SYMBOL_TABLE
"SYS_CBitDB"	DB 2	DB 2	// SYS: Changebit interface
"SYS_DirectCtrlDB"	DB 3	DB 3	// GCS7: PC direct control interface default DB
"SYS_HornDB"	DB 4	DB 4	// GCS7: Data Horn Modul
"SYS_LOG_Queue"	DB 5	DB 5	// PC Interface to log
"GCS7_GrCtrlDBTmp"	DB 6	FB 9	// Class date of FB9
"GCS7_RS485CtrlDB"	DB 7	FB 7	// GCS7: Communication controller opto22
"GCS7_ScaleControlDB"	DB 8	DB 8	// GCS7: Scale control buffer
"GCS7_GrCtrlDB"	DB 9	DB 9	// GCS7: Group control buffer
"SYS_DirectCtrlLCDB"	DB 10	DB 10	// GCS7: PC Direct Control Interface Remote Parameter
"TEST_IOSimuliInput"	DB 16	DB 16	// TEST: Only for serial (MPI) simulation
"TEST_IOSimuliOutput"	DB 17	DB 17	// TEST: Only for serial (MPI) simulation
"KebaHT4Data"	DB 20	FB 80	// Data KebaHT4Data
"SYS_PCCDirectCtrlDB"	DB 40	DB 40	// SYS: PC direct control interface PIC / WinCos /MELE
"SYS_PC1DirectCtrlDB"	DB 41	DB 41	// SYS: PC direct control interface pcc 1 (WinCC)
"SYS_PC2DirectCtrlDB"	DB 42	DB 42	// SYS: PC direct control interface pcc 2 (WinCC)
"SYS_PC3DirectCtrlDB"	DB 43	DB 43	// SYS: PC direct control interface pcc 1 (WinCC)
"SYS_PC4DirectCtrlDB"	DB 44	DB 44	// SYS: PC direct control interface pcc 4 (WinCC)
"SYS_PC5DirectCtrlDB"	DB 45	DB 45	// SYS: PC direct control interface pcc 5 (WinCC)
"SYS_PC6DirectCtrlDB"	DB 46	DB 46	// SYS: PC direct control interface pcc 6 (WinCC)
"SYS_PC7DirectCtrlDB"	DB 47	DB 47	// SYS: PC direct control interface pcc 7 (WinCC)
"SYS_ObjViewDirectCtrlDB"	DB 48	DB 48	// SYS: PC direct control interface for ObjView
"SYS_IHTestDirectCtrlDB"	DB 49	DB 49	// SYS: PC direct control interface for inhouse test
"PLC_SystemDB"	DB 50	DB 50	// PLC: System informations
"PLC_DPInfo"	DB 51	DB 51	// Summary Slave errors
"SSA_SYS_ASI_Info"	DB 52	DB 52	// Summary Slave errors
"PC_StorageDB"	DB 53	DB 53	// PC: Storage with free assignment
"ASW_TimerSettings"	DB 56	DB 56	// ASW: Timer settings
"ASW_Counter"	DB 57	DB 57	// ASW: Counter presettings
"SYS_PC1CBitDB"	DB 61	UDT 10020	// SYS: Changebit interface pcc 1 | PIC.LCT | MELE
"SYS_PC2CBitDB"	DB 62	UDT 10020	// SYS: Changebit interface pcc 2 | PIC.LMX
"SYS_PC3CBitDB"	DB 63	UDT 10020	// SYS: Changebit interface pcc 3
"SYS_PC4CBitDB"	DB 64	UDT 10020	// SYS: Changebit interface pcc 4
"GCS7_EREDB"	DB 71	FB 71	// GCS7: ERE
"SYS_DPInfoM1"	DB 75	FB 76	// SYS: PROFIBUS-DP diagnostic master 1
"SYS_DPInfoM2"	DB 76	FB 76	// SYS: PROFIBUS-DP diagnostic master 2
"SYS_DPInfoM3"	DB 77	FB 76	// SYS: PROFIBUS-DP diagnostic master 3
"SYS_DPInfoM4"	DB 78	FB 76	// SYS: PROFIBUS-DP diagnostic master 4
"PLC_BinListDB"	DB 79	FB 79	// Central bin list DB
"ASW_GraphicData"	DB 80	DB 80
"ASW_PlantParData"	DB 81	DB 81	// Plant parameters and data time
"PCC_Data4"	DB 84	DB 84	// WinCC/PIC
"PCC_Data5"	DB 85	DB 85	// WinCC/PIC
"PCC_Data6"	DB 86	DB 86	// WinCC/PIC
"PCC_Data7"	DB 87	DB 87	// WinCC/PIC
"PCC_Data8"	DB 88	DB 88	// WinCC/PIC
"PCC_Data9"	DB 89	DB 89	// WinCC/PIC
"PCC_YieldScaleDB"	DB 90	DB 90	// PCC: Databuffer for PCC yield calculation
"COM_RS485Loop1DB"	DB 91	FB 7	// COM: RS485 loop1 scales and MYEB
"COM_RS485Loop2DB"	DB 92	FB 7	// COM: RS485 loop2 roolers
"COM_RS485Loop3DB"	DB 93	FB 7	// COM: RS485 loop3
"COM_RS485Loop4DB"	DB 94	FB 7	// COM: RS485 loop4
"SYS_SimpleDPInfo4DB"	DB 98	DB 98	// Data DP Diagnose
"SYS_StartWarningDB"	DB 100	FB 100	// SYS:  Startwarning modul
"G001G"	DB 101	FB 101	// Group-DB  Power supply circuit +C11
"G002G"	DB 102	FB 102	// Group-DB  Contactor panel power supply 1
"G003G"	DB 103	FB 103	// Group-DB  PLC monitoring
"G004G"	DB 104	FB 104	// Group-DB  GENERAL ELEMENTS STEEPING
"G005G"	DB 105	FB 105	// Group-DB  GENERAL ELEMENTS GERM 1
"G006G"	DB 106	FB 106	// Group-DB  GENERAL ELEMENTS GERM 2
"G007G"	DB 107	FB 107	// Group-DB  GENERAL ELEMENTS GERM 3
"G008G"	DB 108	FB 108	// Group-DB  GENERAL ELEMENTS GERM 4
"G009G"	DB 109	FB 109	// Group-DB  GENERAL ELEMENTS GERM 5
"G010G"	DB 110	FB 110	// Group-DB  Line messages
"G011G"	DB 111	FB 111	// Group-DB  MELE/WinCoS communication monitoring
"G012G"	DB 112	FB 112	// Group-DB  GENERAL ELEMENTS GERM 6
"G013G"	DB 113	FB 113	// Group-DB  GENERAL ELEMENTS GERM 7
"G014G"	DB 114	FB 114	// Group-DB  GENERAL ELEMENTS GERM 8
"G015G"	DB 115	FB 115	// Group-DB  CCOMPRESSED AIR PRESSURE STEEP 1 - 4
"G016G"	DB 116	FB 116	// Group-DB  CCOMPRESSED AIR PRESSURE STEEP 5 - 8
"G017G"	DB 117	FB 117	// Group-DB  CCOMPRESSED AIR PRESSURE STEEP 9 - 12
"G018G"	DB 118	FB 118	// Group-DB  CCOMPRESSED AIR PRESSURE STEEP 13 - 16
"G019G"	DB 119	FB 119	// Group-DB  CCOMPRESSED AIR PRESSURE STEEP 17 - 20
"G020G"	DB 120	FB 120	// Group-DB  CCOMPRESSED AIR PRESSURE STEEP 21 - 24
"G021G"	DB 121	FB 121	// Group-DB  GENERAL ELEMENTS KILN 1
"G022G"	DB 122	FB 122	// Group-DB  GENERAL ELEMENTS KILN 2
"G023G"	DB 123	FB 123	// Group-DB  GENERAL ELEMENTS KILN MALT TRANSFER
"G026G"	DB 126	FB 126	// Group-DB  Alarm horns
"G029G"	DB 129	FB 129	// Group-DB  Bin low levels
"G030G"	DB 130	FB 130	// Group-DB  Bin high levels
"G031G"	DB 131	FB 131	// Group-DB  GENERAL ELEMENTS STEEPING
"G032M"	DB 132	FB 132	// Group-DB  CO2 FAN AND FESH AIR FLAP STEEPING 1
"G033M"	DB 133	FB 133	// Group-DB  AERATION AIR STEEPING 1
"G034M"	DB 134	FB 134	// Group-DB  CO2 FAN AND FESH AIR FLAP STEEPING 2
"G035M"	DB 135	FB 135	// Group-DB  AERATION AIR STEEPING 2
"G036M"	DB 136	FB 136	// Group-DB  CO2 FAN AND FESH AIR FLAP STEEPING 3
"G037M"	DB 137	FB 137	// Group-DB  AERATION AIR STEEPING 3
"G038M"	DB 138	FB 138	// Group-DB  CO2 FAN AND FESH AIR FLAP STEEPING 4
"G039M"	DB 139	FB 139	// Group-DB  AERATION AIR STEEPING 4
"G040M"	DB 140	FB 140	// Group-DB  CO2 FAN AND FESH AIR FLAP STEEPING 5
"G041M"	DB 141	FB 141	// Group-DB  AERATION AIR STEEPING 5
"G042M"	DB 142	FB 142	// Group-DB  CO2 FAN AND FESH AIR FLAP STEEPING 6
"G043M"	DB 143	FB 143	// Group-DB  AERATION AIR STEEPING 6
"G044M"	DB 144	FB 144	// Group-DB  CO2 FAN AND FESH AIR FLAP STEEPING 7
"G045M"	DB 145	FB 145	// Group-DB  AERATION AIR STEEPING 7
"G046M"	DB 146	FB 146	// Group-DB  CO2 FAN AND FESH AIR FLAP STEEPING 8
"G047M"	DB 147	FB 147	// Group-DB  AERATION AIR STEEPING 8
"G048M"	DB 148	FB 148	// Group-DB  CO2 FAN AND FESH AIR FLAP STEEPING 9
"G049M"	DB 149	FB 149	// Group-DB  AERATION AIR STEEPING 9
"G050M"	DB 150	FB 150	// Group-DB  CO2 FAN AND FESH AIR FLAP STEEPING 10
"G051M"	DB 151	FB 151	// Group-DB  AERATION AIR STEEPING 10
"G052M"	DB 152	FB 152	// Group-DB  CO2 FAN AND FESH AIR FLAP STEEPING 11
"G053M"	DB 153	FB 153	// Group-DB  AERATION AIR STEEPING 11
"G054M"	DB 154	FB 154	// Group-DB  CO2 FAN AND FESH AIR FLAP STEEPING 12
"G055M"	DB 155	FB 155	// Group-DB  AERATION AIR STEEPING 12
"G056M"	DB 156	FB 156	// Group-DB  CO2 FAN AND FESH AIR FLAP STEEPING 13
"G057M"	DB 157	FB 157	// Group-DB  AERATION AIR STEEPING 13
"G058M"	DB 158	FB 158	// Group-DB  CO2 FAN AND FESH AIR FLAP STEEPING 14
"G059M"	DB 159	FB 159	// Group-DB  AERATION AIR STEEPING 14
"G060M"	DB 160	FB 160	// Group-DB  CO2 FAN AND FESH AIR FLAP STEEPING 15
"G061M"	DB 161	FB 161	// Group-DB  AERATION AIR STEEPING 15
"G062M"	DB 162	FB 162	// Group-DB  CO2 FAN AND FESH AIR FLAP STEEPING 16
"G063M"	DB 163	FB 163	// Group-DB  AERATION AIR STEEPING 16
"G064M"	DB 164	FB 164	// Group-DB  CO2 FAN AND FESH AIR FLAP STEEPING 17
"G065M"	DB 165	FB 165	// Group-DB  AERATION AIR STEEPING 17
"G066M"	DB 166	FB 166	// Group-DB  PRODUCT SLIDER STEEPING 17
"G067M"	DB 167	FB 167	// Group-DB  CO2 FAN AND FESH AIR FLAP STEEPING 18
"G068M"	DB 168	FB 168	// Group-DB  AERATION AIR STEEPING 18
"G069M"	DB 169	FB 169	// Group-DB  PRODUCT SLIDER STEEPING 18
"G070M"	DB 170	FB 170	// Group-DB  CO2 FAN AND FESH AIR FLAP STEEPING 19
"G071M"	DB 171	FB 171	// Group-DB  AERATION AIR STEEPING 19
"G072M"	DB 172	FB 172	// Group-DB  PRODUCT SLIDER STEEPING 19
"G073M"	DB 173	FB 173	// Group-DB  CO2 FAN AND FESH AIR FLAP STEEPING 20
"G074M"	DB 174	FB 174	// Group-DB  AERATION AIR STEEPING 20
"G075M"	DB 175	FB 175	// Group-DB  PRODUCT SLIDER STEEPING 20
"G076M"	DB 176	FB 176	// Group-DB  CO2 FAN AND FESH AIR FLAP STEEPING 21
"G077M"	DB 177	FB 177	// Group-DB  AERATION AIR STEEPING 21
"G078M"	DB 178	FB 178	// Group-DB  PRODUCT SLIDER STEEPING 21
"G079M"	DB 179	FB 179	// Group-DB  CO2 FAN AND FESH AIR FLAP STEEPING 22
"G080M"	DB 180	FB 180	// Group-DB  AERATION AIR STEEPING 22
"G081M"	DB 181	FB 181	// Group-DB  PRODUCT SLIDER STEEPING 22
"G082M"	DB 182	FB 182	// Group-DB  CO2 FAN AND FESH AIR FLAP STEEPING 23
"G083M"	DB 183	FB 183	// Group-DB  AERATION AIR STEEPING 23
"G084M"	DB 184	FB 184	// Group-DB  PRODUCT SLIDER STEEPING 23
"G085M"	DB 185	FB 185	// Group-DB  CO2 FAN AND FESH AIR FLAP STEEPING 24
"G086M"	DB 186	FB 186	// Group-DB  AERATION AIR STEEPING 24
"G087M"	DB 187	FB 187	// Group-DB  PRODUCT SLIDER STEEPING 24
"G090G"	DB 190	FB 190	// Group-DB  GENERAL ELEMENTS GERM 1
"G091M"	DB 191	FB 191	// Group-DB  BELT CONVEYOR 4100 GERM 1-4
"G092M"	DB 192	FB 192	// Group-DB  BELT CONVEYOR 4200 GERM 5-8
"G093M"	DB 193	FB 193	// Group-DB  BELT CONVEYOR 4300 GERM
"G094M"	DB 194	FB 194	// Group-DB  BELT CONVEYOR 4400 GERM
"G095M"	DB 195	FB 195	// Group-DB  BELT CONVEYOR 4500 GERM
"G097M"	DB 197	FB 197	// Group-DB  LIFTING DEVICE GERM 1
"G098M"	DB 198	FB 198	// Group-DB  COUPLING DEVICE TURNER GERM 1
"G099M"	DB 199	FB 199	// Group-DB  COUPLING DEVICE WALL GERM 1
"G100M"	DB 200	FB 200	// Group-DB  TRAVELLING DRIVE GERM 1
"G101M"	DB 201	FB 201	// Group-DB  HORIZONTAL AND LIFTING SCREW GERM 1
"G102M"	DB 202	FB 202	// Group-DB  LOCAL COMMAND BUTTON / LAMPS GERM 1
"G103M"	DB 203	FB 203	// Group-DB  TEMPERATURE MES. GERM 1
"G104M"	DB 204	FB 204	// Group-DB  TURNING SCREWS GERM 1
"G105M"	DB 205	FB 205	// Group-DB  FAN AND VALVE SRAY AIR GERM 1
"G106M"	DB 206	FB 206	// Group-DB  FRESH AIR LOUVER GERM 1
"G107M"	DB 207	FB 207	// Group-DB  EXHAUST AIR LOUVER GERM 1
"G108M"	DB 208	FB 208	// Group-DB  PRODUCT MOISTERING  GERM 1
"G109M"	DB 209	FB 209	// Group-DB  HP CLEANING GERM 1
"G110M"	DB 210	FB 210	// Group-DB  INLET SLIDE GERM 1
"G111M"	DB 211	FB 211	// Group-DB  LOADING CONVEYOR 4600 GERM 1
"G112M"	DB 212	FB 212	// Group-DB  COOLING / HEATING GERM 1
"G113M"	DB 213	FB 213	// Group-DB  BELT CONVEYOR 7050 GERM 1 / 2
"G114M"	DB 214	FB 214	// Group-DB  CHAIN CONVEYOR 7100 GERM
"G120G"	DB 220	FB 220	// Group-DB  GENERAL ELEMENTS GERM 2
"G121M"	DB 221	FB 221	// Group-DB  CHAIN CONVEYOR 4600 GERM 2
"G122M"	DB 222	FB 222	// Group-DB  LIFTING DEVICE GERM 2
"G123M"	DB 223	FB 223	// Group-DB  COUPLING DEVICE TURNER GERM 2
"G124M"	DB 224	FB 224	// Group-DB  COUPLING DEVICE WALL GERM 2
"G125M"	DB 225	FB 225	// Group-DB  TRAVELLING DRIVE GERM 2
"G126M"	DB 226	FB 226	// Group-DB  HORIZONTAL AND LIFTING SCREW GERM 2
"G127M"	DB 227	FB 227	// Group-DB  LOCAL COMMAND BUTTON / LAMPS GERM 2
"G128M"	DB 228	FB 228	// Group-DB  TEMPERATURE MES. GERM 2
"G129M"	DB 229	FB 229	// Group-DB  TURNING SCREWS GERM 2
"G130M"	DB 230	FB 230	// Group-DB  FAN AND VALVE SRAY AIR GERM 2
"G131M"	DB 231	FB 231	// Group-DB  FRESH AIR LOUVER GERM 2
"G132M"	DB 232	FB 232	// Group-DB  EXHAUST AIR  LOUVER GERM 2
"G133M"	DB 233	FB 233	// Group-DB  PRODUCT MOISTERING  GERM 2
"G134M"	DB 234	FB 234	// Group-DB  HP CLEANING GERM 2
"G135M"	DB 235	FB 235	// Group-DB  INLET SLIDE GERM 2
"G136M"	DB 236	FB 236	// Group-DB  LOAD / UNLOAD CONVEYOR GERM 2
"G137M"	DB 237	FB 237	// Group-DB  COOLING / HEATING GERM 2
"G140G"	DB 240	FB 240	// Group-DB  GENERAL ELEMENTS GERM 3
"G141M"	DB 241	FB 241	// Group-DB  CHAIN CONVEYOR 4600 GERM 3
"G142M"	DB 242	FB 242	// Group-DB  LIFTING DEVICE GERM 3
"G143M"	DB 243	FB 243	// Group-DB  COUPLING DEVICE TURNER GERM 3
"G144M"	DB 244	FB 244	// Group-DB  COUPLING DEVICE WALL GERM 3
"G145M"	DB 245	FB 245	// Group-DB  TRAVELLING DRIVE GERM 3
"G146M"	DB 246	FB 246	// Group-DB  HORIZONTAL AND LIFTING SCREW GERM 3
"G147M"	DB 247	FB 247	// Group-DB  LOCAL COMMAND BUTTON / LAMPS GERM 3
"G148M"	DB 248	FB 248	// Group-DB  TEMPERATURE MES. GERM 3
"G149M"	DB 249	FB 249	// Group-DB  TURNING SCREWS GERM 3
"G150M"	DB 250	FB 250	// Group-DB  FAN AND VALVE SRAY AIR GERM 3
"G151M"	DB 251	FB 251	// Group-DB  FRESH AIR LOUVER GERM 3
"G152M"	DB 252	FB 252	// Group-DB  EXHAUST AIR LOUVER GERM 3
"G153M"	DB 253	FB 253	// Group-DB  PRODUCT MOISTERING  GERM 3
"G154M"	DB 254	FB 254	// Group-DB  HP CLEANING GERM 3
"G155M"	DB 255	FB 255	// Group-DB  INLET SLIDE GERM 3
"G156M"	DB 256	FB 256	// Group-DB  LOAD / UNLOAD CONVEYOR GERM 3
"G157M"	DB 257	FB 257	// Group-DB  COOLING / HEATING GERM 3
"G158M"	DB 258	FB 258	// Group-DB  CHAIN CONVEYOR 7050 GERM 3 / 4
"G160G"	DB 260	FB 260	// Group-DB  GENERAL ELEMENTS GERM 4
"G161M"	DB 261	FB 261	// Group-DB  CHAIN CONVEYOR 4600 GERM 4
"G162M"	DB 262	FB 262	// Group-DB  LIFTING DEVICE GERM 4
"G163M"	DB 263	FB 263	// Group-DB  COUPLING DEVICE TURNER GERM 4
"G164M"	DB 264	FB 264	// Group-DB  COUPLING DEVICE WALL GERM 4
"G165M"	DB 265	FB 265	// Group-DB  TRAVELLING DRIVE GERM 4
"G166M"	DB 266	FB 266	// Group-DB  HORIZONTAL AND LIFTING SCREW GERM 4
"G167M"	DB 267	FB 267	// Group-DB  LOCAL COMMAND BUTTON / LAMPS GERM 4
"G168M"	DB 268	FB 268	// Group-DB  TEMPERATURE MES. GERM 4
"G169M"	DB 269	FB 269	// Group-DB  TURNING SCREWS GERM 4
"G170M"	DB 270	FB 270	// Group-DB  FAN AND VALVE SRAY AIR GERM 4
"G171M"	DB 271	FB 271	// Group-DB  FRESH AIR LOUVER GERM 4
"G172M"	DB 272	FB 272	// Group-DB  EXHAUST AIR LOUVER GERM 4
"G173M"	DB 273	FB 273	// Group-DB  PRODUCT MOISTERING  GERM 4
"G174M"	DB 274	FB 274	// Group-DB  HP CLEANING GERM 4
"G175M"	DB 275	FB 275	// Group-DB  INLET SLIDE GERM 4
"G176M"	DB 276	FB 276	// Group-DB  LOAD / UNLOAD CONVEYOR GERM 4
"G177M"	DB 277	FB 277	// Group-DB  COOLING / HEATING GERM 4
"G180G"	DB 280	FB 280	// Group-DB  GENERAL ELEMENTS GERM 5
"G181M"	DB 281	FB 281	// Group-DB  CHAIN CONVEYOR 4600 GERM 5
"G182M"	DB 282	FB 282	// Group-DB  LIFTING DEVICE GERM 5
"G183M"	DB 283	FB 283	// Group-DB  COUPLING DEVICE TURNER GERM 5
"G184M"	DB 284	FB 284	// Group-DB  COUPLING DEVICE WALL GERM 5
"G185M"	DB 285	FB 285	// Group-DB  TRAVELLING DRIVE GERM 5
"G186M"	DB 286	FB 286	// Group-DB  HORIZONTAL AND LIFTING SCREW GERM 5
"G187M"	DB 287	FB 287	// Group-DB  LOCAL COMMAND BUTTON / LAMPS GERM 5
"G188M"	DB 288	FB 288	// Group-DB  TEMPERATURE MES. GERM 5
"G189M"	DB 289	FB 289	// Group-DB  TURNING SCREWS GERM 5
"G190M"	DB 290	FB 290	// Group-DB  FAN AND VALVE SRAY AIR GERM 5
"G191M"	DB 291	FB 291	// Group-DB  FRESH AIR LOUVER GERM 5
"G192M"	DB 292	FB 292	// Group-DB  EXHAUST AIR LOUVER GERM 5
"G193M"	DB 293	FB 293	// Group-DB  PRODUCT MOISTERING  GERM 5
"G194M"	DB 294	FB 294	// Group-DB  HP CLEANING GERM 5
"G195M"	DB 295	FB 295	// Group-DB  INLET SLIDE GERM 5
"G196M"	DB 296	FB 296	// Group-DB  LOAD / UNLOAD CONVEYOR GERM 5
"G197M"	DB 297	FB 297	// Group-DB  COOLING / HEATING GERM 5
"G198M"	DB 298	FB 298	// Group-DB  CHAIN CONVEYOR 7050 GERM 5 / 6
"G200G"	DB 300	FB 300	// Group-DB  GENERAL ELEMENTS GERM 6
"G201M"	DB 301	FB 301	// Group-DB  CHAIN CONVEYOR 4600 GERM 6
"G202M"	DB 302	FB 302	// Group-DB  LIFTING DEVICE GERM 6
"G203M"	DB 303	FB 303	// Group-DB  COUPLING DEVICE TURNER GERM 6
"G204M"	DB 304	FB 304	// Group-DB  COUPLING DEVICE WALL GERM 6
"G205M"	DB 305	FB 305	// Group-DB  TRAVELLING DRIVE GERM 6
"G206M"	DB 306	FB 306	// Group-DB  HORIZONTAL AND LIFTING SCREW GERM 6
"G207M"	DB 307	FB 307	// Group-DB  LOCAL COMMAND BUTTON / LAMPS GERM 6
"G208M"	DB 308	FB 308	// Group-DB  TEMPERATURE MES. GERM 6
"G209M"	DB 309	FB 309	// Group-DB  TURNING SCREWS GERM 6
"G210M"	DB 310	FB 310	// Group-DB  FAN AND VALVE SRAY AIR GERM 6
"G211M"	DB 311	FB 311	// Group-DB  FRESH AIR LOUVER GERM 6
"G212M"	DB 312	FB 312	// Group-DB  EXHAUST AIR LOUVER GERM 6
"G213M"	DB 313	FB 313	// Group-DB  PRODUCT MOISTERING  GERM 6
"G214M"	DB 314	FB 314	// Group-DB  HP CLEANING GERM 6
"G215M"	DB 315	FB 315	// Group-DB  INLET SLIDE GERM 6
"G216M"	DB 316	FB 316	// Group-DB  LOAD / UNLOAD CONVEYOR GERM 6
"G217M"	DB 317	FB 317	// Group-DB  COOLING / HEATING GERM 6
"G220G"	DB 320	FB 320	// Group-DB  GENERAL ELEMENTS GERM 7
"G221M"	DB 321	FB 321	// Group-DB  CHAIN CONVEYOR 4600 GERM 7
"G222M"	DB 322	FB 322	// Group-DB  LIFTING DEVICE GERM 7
"G223M"	DB 323	FB 323	// Group-DB  COUPLING DEVICE TURNER GERM 7
"G224M"	DB 324	FB 324	// Group-DB  COUPLING DEVICE WALL GERM 7
"G225M"	DB 325	FB 325	// Group-DB  TRAVELLING DRIVE GERM 7
"G226M"	DB 326	FB 326	// Group-DB  HORIZONTAL AND LIFTING SCREW GERM 7
"G227M"	DB 327	FB 327	// Group-DB  LOCAL COMMAND BUTTON / LAMPS GERM 7
"G228M"	DB 328	FB 328	// Group-DB  TEMPERATURE MES. GERM 7
"G229M"	DB 329	FB 329	// Group-DB  TURNING SCREWS GERM 7
"G230M"	DB 330	FB 330	// Group-DB  FAN AND VALVE SRAY AIR GERM 7
"G231M"	DB 331	FB 331	// Group-DB  FRESH AIR LOUVER GERM 7
"G232M"	DB 332	FB 332	// Group-DB  EXHAUST AIR LOUVER GERM 7
"G233M"	DB 333	FB 333	// Group-DB  PRODUCT MOISTERING  GERM 7
"G234M"	DB 334	FB 334	// Group-DB  HP CLEANING GERM 7
"G235M"	DB 335	FB 335	// Group-DB  INLET SLIDE GERM 7
"G236M"	DB 336	FB 336	// Group-DB  LOAD / UNLOAD CONVEYOR GERM 7
"G237M"	DB 337	FB 337	// Group-DB  COOLING / HEATING GERM 7
"G238M"	DB 338	FB 338	// Group-DB  CHAIN CONVEYOR 7050 GERM 7 / 8
"G240G"	DB 340	FB 340	// Group-DB  GENERAL ELEMENTS GERM 8
"G241M"	DB 341	FB 341	// Group-DB  CHAIN CONVEYOR 4600 GERM 8
"G242M"	DB 342	FB 342	// Group-DB  LIFTING DEVICE GERM 8
"G243M"	DB 343	FB 343	// Group-DB  COUPLING DEVICE TURNER GERM 8
"G244M"	DB 344	FB 344	// Group-DB  COUPLING DEVICE WALL GERM 8
"G245M"	DB 345	FB 345	// Group-DB  TRAVELLING DRIVE GERM 8
"G246M"	DB 346	FB 346	// Group-DB  HORIZONTAL AND LIFTING SCREW GERM 8
"G247M"	DB 347	FB 347	// Group-DB  LOCAL COMMAND BUTTON / LAMPS GERM 8
"G248M"	DB 348	FB 348	// Group-DB  TEMPERATURE MES. GERM 8
"G249M"	DB 349	FB 349	// Group-DB  TURNING SCREWS GERM 8
"G250M"	DB 350	FB 350	// Group-DB  FAN AND VALVE SRAY AIR GERM 8
"G251M"	DB 351	FB 351	// Group-DB  FRESH AIR LOUVER GERM 8
"G252M"	DB 352	FB 352	// Group-DB  EXHAUST AIR LOUVER GERM 8
"G253M"	DB 353	FB 353	// Group-DB  PRODUCT MOISTERING  GERM 8
"G254M"	DB 354	FB 354	// Group-DB  HP CLEANING GERM 8
"G255M"	DB 355	FB 355	// Group-DB  INLET SLIDE GERM 8
"G256M"	DB 356	FB 356	// Group-DB  LOAD / UNLOAD CONVEYOR GERM 8
"G257M"	DB 357	FB 357	// Group-DB  COOLING / HEATING GERM 8
"G260G"	DB 360	FB 360	// Group-DB  GENERAL ELEMENTS KILN 1
"G261M"	DB 361	FB 361	// Group-DB  BELT CONVEYOR 7200 KILN
"G262M"	DB 362	FB 362	// Group-DB  BELT CONVEYOR 7300 KILN
"G263M"	DB 363	FB 363	// Group-DB  BELT CONVEYOR 7301 KILN
"G264M"	DB 364	FB 364	// Group-DB  BELT CONVEYOR 7400 KILN
"G265M"	DB 365	FB 365	// Group-DB  LIFTING DEVICE KILN 1
"G266M"	DB 366	FB 366	// Group-DB  TRAVELLING DRIVE KILN 1
"G267M"	DB 367	FB 367	// Group-DB  UNLOADING / LOADING SCREW KILN 1
"G268M"	DB 368	FB 368	// Group-DB  DISCHARGE DOOR KILN 1
"G269M"	DB 369	FB 369	// Group-DB  TEMPERATURE MES. KILN 1
"G270M"	DB 370	FB 370	// Group-DB  AIR SHUT SLIDE KILN 1
"G271M"	DB 371	FB 371	// Group-DB  FAN KILN 1
"G272M"	DB 372	FB 372	// Group-DB  FRESH AIR RECYCLING KILN 1
"G273M"	DB 373	FB 373	// Group-DB  RECYCLING AIR LOUVER KILN 1
"G274M"	DB 374	FB 374	// Group-DB  EXHAUST AIR LOUVER KILN 1
"G275M"	DB 375	FB 375	// Group-DB  BYPASS FLAP KILN 1
"G276M"	DB 376	FB 376	// Group-DB  HEATING KILN 1
"G277M"	DB 377	FB 377	// Group-DB  LOUVER AIR HEATER KILN 1
"G278M"	DB 378	FB 378	// Group-DB  WITHERING AIR KILN 1
"G279M"	DB 379	FB 379	// Group-DB  HEATING KILN 1 + 2
"G280M"	DB 380	FB 380	// Group-DB  CHAIN CONVEYOR 9001 KILN 1
"G281M"	DB 381	FB 381	// Group-DB  ELEVATOR 9002 AFTER KILN
"G282M"	DB 382	FB 382	// Group-DB  FLAP BOX 9008
"G283M"	DB 383	FB 383	// Group-DB  CULM BATCH BIN 9005
"G284M"	DB 384	FB 384	// Group-DB  BELT CONVEYOR 7100 KILN
"G290G"	DB 390	FB 390	// Group-DB  GENERAL ELEMENTS KILN 2
"G291M"	DB 391	FB 391	// Group-DB  LIFTING DEVICE KILN 2
"G292M"	DB 392	FB 392	// Group-DB  TRAVELLING DRIVE KILN 2
"G293M"	DB 393	FB 393	// Group-DB  UNLOADING / LOADING SCREW KILN 2
"G294M"	DB 394	FB 394	// Group-DB  DISCHARGE DOOR KILN 2
"G295M"	DB 395	FB 395	// Group-DB  TEMPERATURE MES. KILN 2
"G296M"	DB 396	FB 396	// Group-DB  AIR SHUT SLIDE KILN 2
"G297M"	DB 397	FB 397	// Group-DB  FAN KILN 2
"G298M"	DB 398	FB 398	// Group-DB  FRESH AIR FLAP KILN 2
"G299M"	DB 399	FB 399	// Group-DB  RECYCLING AIR FLAP KILN 2
"G300M"	DB 400	FB 400	// Group-DB  EXHAUST AIR FLAP KILN 2
"G301M"	DB 401	FB 401	// Group-DB  BYPASS FLAP KILN 2
"G302M"	DB 402	FB 402	// Group-DB  HEATING KILN 2
"G303M"	DB 403	FB 403	// Group-DB  LOUVER AIR HEATER KILN 2
"G304M"	DB 404	FB 404	// Group-DB  WITHERING AIR KILN 2
"G305M"	DB 405	FB 405	// Group-DB  CHAIN CONVEYOR 9002 KILN 2
"G306M"	DB 406	FB 406	// Group-DB  DMBG DISCHARGER KILN MALT TRANSFER
"G307M"	DB 407	FB 407	// Group-DB  SCREW CONVEYOR 9007 KILN MALT TRANSFER
"G308M"	DB 408	FB 408	// Group-DB  BELT CONVEYOR 9009 KILN MALT TRANSFER
"G309M"	DB 409	FB 409	// Group-DB  ELEVATOR EXCISTING
"G310M"	DB 410	FB 410	// Group-DB  PLC1 TO EXCISTING DEGERMINATION SYSTEM
"G311M"	DB 411	FB 411	// Group-DB  CENTRAL ASPIRATION UNLOAD KILN
"G320M"	DB 420	FB 420	// Group-DB  PCC GRAPHIC SUPPORT
"EventsToPIC_DB"	DB 470	FB 470
"ASW_DFCATargData"	DB 480	DB 480	// ASW_DFCATargData
"INT1S001SND33"	DB 515	DB 515	// Bin DB  Wheat intake sender
"INT1S001RCV34"	DB 516	DB 516	// Bin DB  Wheat intake receiver
"FCL1S001SND33"	DB 535	DB 535	// Bin DB  1st cleaning sender
"FCL1S001RCV34"	DB 536	DB 536	// Bin DB  1st cleaning receiver
"SDP1S001SND33"	DB 545	DB 545	// Bin DB  2nd dampening sender
"SDP1S001RCV34"	DB 546	DB 546	// Bin DB  2nd dampening receiver
"SCL1S001SND33"	DB 555	DB 555	// Bin DB  2nd cleaning sender
"SCL1S001RCV34"	DB 556	DB 556	// Bin DB  2nd cleaning receiver
"FTR1S001SND33"	DB 575	DB 575	// Bin DB  Flour transfer sender
"FTR1S001RCV34"	DB 576	DB 576	// Bin DB  Flour transfer receiver
"OTL1S001SND33"	DB 585	DB 585	// Bin DB  Flour bulk outload sender
"OTL1S001RCV34"	DB 586	DB 586	// Bin DB  Flour bulk outload receiver
"SCG1S001SND33"	DB 595	DB 595	// Bin DB  Screenings grinding sender
"SCG1S001RCV34"	DB 596	DB 596	// Bin DB  Screenings grinding receiver
"BTR1S001SND33"	DB 605	DB 605	// Bin DB  Bran turnover sender
"BTR1S001RCV34"	DB 606	DB 606	// Bin DB  Bran turnover receiver
"MAL1Par"	DB 799	DB 799	// Line parameter data block
"MAL1"	DB 800	DB 800	// Line data block  MALTING LINE
"MAL1S001"	DB 801	DB 801	// Section data block  LINE 1 SEC 1 SECTIONDATA
"MAL1S005"	DB 805	DB 805	// Section data block  STEEPING ROW 1 (ST1-8)
"MAL1S006"	DB 806	DB 806	// Section data block  STEEPING ROW 2 (ST9-16)
"MAL1S007"	DB 807	DB 807	// Section data block  STEEPING ROW 3 (ST17-24)
"MAL1S017"	DB 817	DB 817	// Section data block  LINE 1 SEC 17 GERM 1
"MAL1S018"	DB 818	DB 818	// Section data block  LINE 1 SEC 18 GERM 2
"MAL1S019"	DB 819	DB 819	// Section data block  LINE 1 SEC 19 GERM 3
"MAL1S020"	DB 820	DB 820	// Section data block  LINE 1 SEC 20 GERM 4
"MAL1S021"	DB 821	DB 821	// Section data block  LINE 1 SEC 21 GERM 5
"MAL1S022"	DB 822	DB 822	// Section data block  LINE 1 SEC 22 GERM 6
"MAL1S023"	DB 823	DB 823	// Section data block  LINE 1 SEC 23 GERM 7
"MAL1S024"	DB 824	DB 824	// Section data block  LINE 1 SEC 24 GERM 8
"MAL1S032"	DB 832	DB 832	// Section data block  LINE 1 SEC 32 KILN 1
"MAL1S033"	DB 833	DB 833	// Section data block  LINE 1 SEC 33 KILN 2
"MAL1S034"	DB 834	DB 834	// Section data block  LINE 1 SEC 34 UNLOAD KILN
"MAL1S001SND33"	DB 843	DB 843	// Bin DB  Dummy sender
"MAL1S001RCV34"	DB 844	DB 844	// Bin DB  Dummy receiver
"MAl1S034SND35"	DB 845	DB 845	// Bin DB  KILNED MALT BINS
"MAl1S034RCV36"	DB 846	DB 846	// Bin DB  KILNED MALT BINS
"MAL1S005Par"	DB 895	DB 895	// Parameter data block  STEEPING ROW 1 (ST1-8)
"MAL1S006Par"	DB 896	DB 896	// Parameter data block  STEEPING ROW 2 (ST9-16)
"MAL1S007Par"	DB 897	DB 897	// Parameter data block  STEEPING ROW 3 (ST17-24)
"MAL1S005_ST1Par"	DB 900	DB 900	// Parameter data block  STEEPING ROW 1 (ST1-8)
"MAL1S017Par"	DB 907	DB 907	// Parameter data block  LINE 1 SEC 17 GERM 1
"MAL1S018Par"	DB 908	DB 908	// Parameter data block  LINE 1 SEC 18 GERM 2
"MAL1S019Par"	DB 909	DB 909	// Parameter data block  LINE 1 SEC 19 GERM 3
"MAL1S020Par"	DB 910	DB 910	// Parameter data block  LINE 1 SEC 20 GERM 4
"MAL1S021Par"	DB 911	DB 911	// Parameter data block  LINE 1 SEC 21 GERM 5
"MAL1S022Par"	DB 912	DB 912	// Parameter data block  LINE 1 SEC 22 GERM 6
"MAL1S023Par"	DB 913	DB 913	// Parameter data block  LINE 1 SEC 23 GERM 7
"MAL1S024Par"	DB 914	DB 914	// Parameter data block  LINE 1 SEC 24 GERM 8
"MAL1S032Par"	DB 922	DB 922	// Parameter data block  LINE 1 SEC 32 KILN 1
"MAL1S033Par"	DB 923	DB 923	// Parameter data block  LINE 1 SEC 33 KILN 2
"SSA_LOG_Value_Queue"	DB 1005	DB 1005	// PC Interface to log
"MAL1ProcessTime"	DB 1013	DB 1013	// ProcessTime  MALTING LINE
"PLC1Snd"	DB 1711	DB 1711	// COM: Send data to PLC 1
"PLC2Snd"	DB 1712	DB 1712	// COM: Send data to PLC 2
"PLC3Snd"	DB 1713	DB 1713	// COM: Send data to PLC 3
"PLC4Snd"	DB 1714	DB 1714	// COM: Send data to PLC 4
"PLC5Snd"	DB 1715	DB 1715	// COM: Send data to PLC 5
"PLC6Snd"	DB 1716	DB 1716	// COM: Send data to PLC 6
"PLC7Snd"	DB 1717	DB 1717	// COM: Send data to PLC 7
"PLC8Snd"	DB 1718	DB 1718	// COM: Send data to PLC 8
"PLC9Snd"	DB 1719	DB 1719	// COM: Send data to PLC 9
"PLC1Rcv"	DB 1721	DB 1721	// COM: Receive data from PLC 1
"PLC2Rcv"	DB 1722	DB 1722	// COM: Receive data from PLC 2
"PLC3Rcv"	DB 1723	DB 1723	// COM: Receive data from PLC 3
"PLC4Rcv"	DB 1724	DB 1724	// COM: Receive data from PLC 4
"PLC5Rcv"	DB 1725	DB 1725	// COM: Receive data from PLC 5
"PLC6Rcv"	DB 1726	DB 1726	// COM: Receive data from PLC 6
"PLC7Rcv"	DB 1727	DB 1727	// COM: Receive data from PLC 7
"PLC8Rcv"	DB 1728	DB 1728	// COM: Receive data from PLC 8
"PLC9Rcv"	DB 1729	DB 1729	// COM: Receive data from PLC 9
"PLC10Snd"	DB 1730	DB 1730	// COM: Send data to PLC 10
"PLC11Snd"	DB 1731	DB 1731	// COM: Send data to PLC 11
"PLC12Snd"	DB 1732	DB 1732	// COM: Send data to PLC 12
"PLC13Snd"	DB 1733	DB 1733	// COM: Send data to PLC 13
"PLC14Snd"	DB 1734	DB 1734	// COM: Send data to PLC 14
"PLC15Snd"	DB 1735	DB 1735	// COM: Send data to PLC 15
"PLC16Snd"	DB 1736	DB 1736	// COM: Send data to PLC 16
"PLC10Rcv"	DB 1740	DB 1740	// COM: Receive data from PLC 10
"PLC11Rcv"	DB 1741	DB 1741	// COM: Receive data from PLC 11
"PLC12Rcv"	DB 1742	DB 1742	// COM: Receive data from PLC 12
"PLC13Rcv"	DB 1743	DB 1743	// COM: Receive data from PLC 13
"PLC14Rcv"	DB 1744	DB 1744	// COM: Receive data from PLC 14
"PLC15Rcv"	DB 1745	DB 1745	// COM: Receive data from PLC 15
"PLC16Rcv"	DB 1746	DB 1746	// COM: Receive data from PLC 16
"ComPLC1Snd"	DB 1761	FB 1701	// COM: Send buffer PLC 1
"ComPLC2Snd"	DB 1762	FB 1701	// COM: Send buffer PLC 2
"ComPLC3Snd"	DB 1763	FB 1701	// COM: Send buffer PLC 3
"ComPLC4Snd"	DB 1764	FB 1701	// COM: Send buffer PLC 4
"ComPLC5Snd"	DB 1765	FB 1701	// COM: Send buffer PLC 5
"ComPLC6Snd"	DB 1766	FB 1701	// COM: Send buffer PLC 6
"ComPLC7Snd"	DB 1767	FB 1701	// COM: Send buffer PLC 7
"ComPLC8Snd"	DB 1768	FB 1701	// COM: Send buffer PLC 8
"ComPLC9Snd"	DB 1769	FB 1701	// COM: Send buffer PLC 9
"ComPLC1Rcv"	DB 1771	FB 1702	// COM: Receive buffer PLC 1
"ComPLC2Rcv"	DB 1772	FB 1702	// COM: Receive buffer PLC 2
"ComPLC3Rcv"	DB 1773	FB 1702	// COM: Receive buffer PLC 3
"ComPLC4Rcv"	DB 1774	FB 1702	// COM: Receive buffer PLC 4
"ComPLC5Rcv"	DB 1775	FB 1702	// COM: Receive buffer PLC 5
"ComPLC6Rcv"	DB 1776	FB 1702	// COM: Receive buffer PLC 6
"ComPLC7Rcv"	DB 1777	FB 1702	// COM: Receive buffer PLC 7
"ComPLC8Rcv"	DB 1778	FB 1702	// COM: Receive buffer PLC 8
"ComPLC9Rcv"	DB 1779	FB 1702	// COM: Receive buffer PLC 9
"ComPLC10Snd"	DB 1780	FB 1701	// COM: Send buffer PLC 10
"ComPLC11Snd"	DB 1781	FB 1701	// COM: Send buffer PLC 11
"ComPLC12Snd"	DB 1782	FB 1701	// COM: Send buffer PLC 12
"ComPLC13Snd"	DB 1783	FB 1701	// COM: Send buffer PLC 13
"ComPLC14Snd"	DB 1784	FB 1701	// COM: Send buffer PLC 14
"ComPLC15Snd"	DB 1785	FB 1701	// COM: Send buffer PLC 15
"ComPLC16Snd"	DB 1786	FB 1701	// COM: Send buffer PLC 16
"ComPLC10Rcv"	DB 1790	FB 1702	// COM: Receive buffer PLC 7
"ComPLC11Rcv"	DB 1791	FB 1702	// COM: Receive buffer PLC 1
"ComPLC12Rcv"	DB 1792	FB 1702	// COM: Receive buffer PLC 2
"ComPLC13Rcv"	DB 1793	FB 1702	// COM: Receive buffer PLC 3
"ComPLC14Rcv"	DB 1794	FB 1702	// COM: Receive buffer PLC 4
"ComPLC15Rcv"	DB 1795	FB 1702	// COM: Receive buffer PLC 5
"ComPLC16Rcv"	DB 1796	FB 1702	// COM: Receive buffer PLC 6
"MAL1S005StepValues"	DB 2005	FB 472	// Data block for Log of Step Values STEEPING ROW 1 (ST1-8)
"MAL1S006StepValues"	DB 2006	FB 472	// Data block for Log of Step Values STEEPING ROW 2 (ST9-16)
"MAL1S007StepValues"	DB 2007	FB 472	// Data block for Log of Step Values STEEPING ROW 3 (ST17-24)
"SSA_VIS_Filter"	DB 2010	DB 2010	// Filter DB to convert Status for Viscontrol
"MAL1S017StepValues"	DB 2017	FB 472	// Data block for Log of Step Values LINE 1 SEC 17 GERM 1
"MAL1S018StepValues"	DB 2018	FB 472	// Data block for Log of Step Values LINE 1 SEC 18 GERM 2
"MAL1S019StepValues"	DB 2019	FB 472	// Data block for Log of Step Values LINE 1 SEC 19 GERM 3
"MAL1S020StepValues"	DB 2020	FB 472	// Data block for Log of Step Values LINE 1 SEC 20 GERM 4
"MAL1S021StepValues"	DB 2021	FB 472	// Data block for Log of Step Values LINE 1 SEC 21 GERM 5
"MAL1S022StepValues"	DB 2022	FB 472	// Data block for Log of Step Values LINE 1 SEC 22 GERM 6
"MAL1S023StepValues"	DB 2023	FB 472	// Data block for Log of Step Values LINE 1 SEC 23 GERM 7
"MAL1S024StepValues"	DB 2024	FB 472	// Data block for Log of Step Values LINE 1 SEC 24 GERM 8
"MAL1S005_ST1Event"	DB 2030	FB 470	// Event data block  STEEPING ROW 1 (ST1-8)
"MAL1S032StepValues"	DB 2032	FB 472	// Data block for Log of Step Values LINE 1 SEC 32 KILN 1
"MAL1S033StepValues"	DB 2033	FB 472	// Data block for Log of Step Values LINE 1 SEC 33 KILN 2
"MAL1S005Event"	DB 2035	FB 470	// Event data block  STEEPING ROW 1 (ST1-8)
"MAL1S006Event"	DB 2036	FB 470	// Event data block  STEEPING ROW 2 (ST9-16)
"MAL1S007Event"	DB 2037	FB 470	// Event data block  STEEPING ROW 3 (ST17-24)
"MAL1S017Event"	DB 2047	FB 470	// Event data block  LINE 1 SEC 17 GERM 1
"MAL1S018Event"	DB 2048	FB 470	// Event data block  LINE 1 SEC 18 GERM 2
"MAL1S019Event"	DB 2049	FB 470	// Event data block  LINE 1 SEC 19 GERM 3
"MAL1S020Event"	DB 2050	FB 470	// Event data block  LINE 1 SEC 20 GERM 4
"MAL1S021Event"	DB 2051	FB 470	// Event data block  LINE 1 SEC 21 GERM 5
"MAL1S022Event"	DB 2052	FB 470	// Event data block  LINE 1 SEC 22 GERM 6
"MAL1S023Event"	DB 2053	FB 470	// Event data block  LINE 1 SEC 23 GERM 7
"MAL1S024Event"	DB 2054	FB 470	// Event data block  LINE 1 SEC 24 GERM 8
"MAL1S032Event"	DB 2062	FB 470	// Event data block  LINE 1 SEC 32 KILN 1
"MAL1S033Event"	DB 2063	FB 470	// Event data block  LINE 1 SEC 33 KILN 2
"SIEMENS_READ"	FB 3	FB 3	// SIEMENS: FMS.read services with SIMATIC NET CPs
"SIEMENS_WRITE"	FB 6	FB 6	// SIEMENS: FMS.write services with SIMATIC NET CPs
"GCS7_RS485Ctrl"	FB 7	FB 7	// GCS7: Communication controller opto22
"GCS7_GrpCtrlMain"	FB 9	FB 9	// GCS7: Group control main program
"GCS7_GrpCtrlSub"	FB 10	FB 10	// GCS7: Group control subroutines
"GCS7_E_DigOutput"	FB 11	FB 11	// GCS7: Element digital output
"GCS7_E_Motor"	FB 12	FB 12	// GCS7: Element motor
"GCS7_E_ValveControl"	FB 13	FB 13	// GCS7: Element valve control
"GCS7_E_DigInput"	FB 14	FB 14	// GCS7: Element digital input continuous
"GCS7_E_PressureRange"	FB 16	FB 16	// GCS7: Element pressure range
"GCS7_E_AnalogOutput"	FB 17	FB 17	// GCS7: Element analog output
"GCS7_E_ATV"	FB 18	FB 18	// Element Control FU Altivar with Profibus
"GCS7_E_AnalogInput"	FB 19	FB 19	// GCS7: Element analog input
"GCS7_E_ValveControl4Pos"	FB 20	FB 20	// GCS7: Element valve control with 4 positions
"GCS7_E_DMDS"	FB 21	FB 21	// GCS7: Element DMDS
"GCS7_E_MZMN"	FB 22	FB 22	// GCS7: Element MZMN micro dosing
"GCS7_E_MYEB"	FB 23	FB 23	// GCS7: Element MYEB moisture control unit
"GCS7_E_MOZE"	FB 24	FB 24	// GCS7: Element MOZE water doser
"GCS7_E_MessageCtrl"	FB 25	FB 25	// GCS7: Element Control Message
"GCS7_E_DFCO"	FB 26	FB 26
"GCS7_E_MEAF_Bag"	FB 27	FB 27	// GCS7: Element Control MEAF-Bag with DP or OPTO22
"GCS7_E_FBAL"	FB 28	FB 28	// GCS7: Element Control Message
"GCS7_E_Sampler"	FB 29	FB 29	// GCS7: Element sampler MZER
"GCS7_E_Maintanance1"	FB 30	FB 30	// GCS7: Element Control Message
"GCS7_E_Maintanance2"	FB 31	FB 31	// GCS7: Element Control Message
"GCS7_E_MZAF"	FB 32	FB 32	// GCS7: Element MZAF flowbalancer
"GCS7_E_MYAH"	FB 33	FB 33	// GCS7: Element MYAH Yield PC
"GCS7_E_MYFC_MOZF"	FB 34	FB 34	// GCS7: Element MYFC/MOZF
"GCS7_E_MDDx"	FB 35	FB 35	// GCS7 Element MDDx Opto22 Communication
"GCS7_E_MYRA_MDEx"	FB 36	FB 36	// GCS7: Element MYRA/MDEF
"GCS7_E_MDDx_DP"	FB 37	FB 37	// SSW: Element MDDR/T Profibus Communication
"GCS7_E_DEVC"	FB 38	FB 38	// GCS7: Element MEAF Dev Control
"GCS7_E_MYFA_MOZD"	FB 39	FB 39	// GCS7: Element MYFA/MOZD automatic dampener
"GCS7_E_Scale"	FB 40	FB 40	// GCS7: Element scale control MWEE, MWEG,
"GCS7_M_MYFA"	FB 41	FB 41	// GCS7: Machine MYFA
"GCS7_E_BSPB"	FB 42	FB 42	// Vertikalschleifer
"GCS7_E_DCOS"	FB 43	FB 43	// GCS7: Element Control Dosing Control System
"GCS7_M_Scourer"	FB 44	FB 44	// GCS7: Machine scourer MHXF
"GCS7_M_Roll4Stand"	FB 45	FB 45	// GCS7: Machine 4 roll stand
"GCS7_M_Roll8Stand"	FB 46	FB 46	// GCS7: Machine 8 roll stand
"GCS7_M_PelletCooler"	FB 47	FB 47	// GCS7: Machine pellet cooler
"GCS7_M_Motors3W2HL"	FB 48	FB 48	// GCS7: Machine 3 Motors and 2 high levels
"GCS7_M_MDDX"	FB 49	FB 49	// GCS7: Machine Newtronic Roll Stand
"GCS7_M_Motor6Mon"	FB 50	FB 50	// GCS7: Machine motor with 6 monitoring elements
"GCS7_M_Motor2Mon"	FB 51	FB 51	// GCS7: Machine motor with 2 monitoring elements
"GCS7_M_MotorBypass"	FB 52	FB 52	// GCS7: Machine motor with bypass
"GCS7_M_Hopper"	FB 53	FB 53	// GCS7: Machine hopper
"GCS7_M_Mixer"	FB 54	FB 54	// GCS7: Machine mixer
"GCS7_M_DFZK"	FB 55	FB 55	// GCS7 Machine DFZK Vertical Rotor Mill
"GCS7_M_Discharger"	FB 56	FB 56	// GCS7: Machine discharger A
"GCS7_E_MTRI"	FB 57	FB 57	// GCS7: Element MTRI Remote Control
"GCS7_M_BCFA"	FB 58	FB 58	// GCS7: Machine Flaker Control System
"GCS7_M_DischargerMZAx"	FB 59	FB 59	// GCS7: Machine discharger with MZAF
"GCS7_M_Aspiration"	FB 60	FB 60	// GCS7: Machine aspiration
"GCS7_M_DPScaleMWBL_MWBS"	FB 61	FB 61	// GCS7: Machine MWBL/MWBS (Profibus+ Opto22)
"GCS7_M_DriveCurrent"	FB 62	FB 62	// GCS7: Machine DriveCurrent
"GCS7_M_DFCA"	FB 63	FB 63	// GCS7: Machine DFCA
"GCS7_M_MYFB"	FB 64	FB 64	// GCS7: Machine MYFB automatic dampener
"GCS7_M_PulsePhaseConv"	FB 65	FB 65	// GCS7: Machine pulse phase conveying system
"GCS7_M_Flift1Airlock"	FB 66	FB 66	// GCS7: Machine fluidlift with 1 airlock
"GCS7_M_Flift2Airlock"	FB 67	FB 67	// GCS7: Machine fluidlift with 2 airlocks
"GCS7_M_PressureVessel"	FB 68	FB 68	// GCS7 Machine Pressure Vessel Conveying
"GCS7_M_RotaryDis"	FB 69	FB 69	// GCS7: Machine rotary distributer
"GCS7_AddWayPattern"	FB 70	FB 70	// GCS7: Old and new waypattern are active
"GCS7_E_MaintananceCnt"	FB 71	FB 71	// GCS7: Maintanance Counter
"GCS7_E_DFCA_Com"	FB 73	FB 73	// GCS7: Communication DFCA pellet press
"GCS7_E_DFCA_Log"	FB 74	FB 74	// GCS7: Log when modify a parameter
"SYS_DP-Diagnosis"	FB 76	FB 76	// SIEMENS_DP-Diagnosis
"GCS7_ULQueue"	FB 77	FB 77
"GCS7_Bin"	FB 78	FB 78	// Functionality of a bin
"PLC_BinList"	FB 79	FB 79	// Central bin list
"KebaHT4"	FB 80	FB 80	// MAINTENANCE MOTOR CONTROL "HT4"
"GCS7_M_RGRP"	FB 81	FB 81	// GCS7: Machine RGRP
"GCS7_M_FluidlifVessel"	FB 82	FB 82	// GCS7 Machine Fluidlift with Pressure Vessel
"GCS7_E_Level"	FB 84	FB 84	// Level: Subtype of FB14
"GCS7_LiftingDevice"	FB 85	FB 85	// de: Hubzug
"GCS7_TractionDrive"	FB 86	FB 86	// Traction drive  de: Fahrantrieb
"GCS7_M_Roll8Stand_DP"	FB 87	FB 87	// SS: Machine 4/8 roll stand wit profibus
"GCS7_Ma_DischagerFlat"	FB 88	FB 88	// Machine Flat-bottom discharger
"STD_LineSecStdSub2"	FB 90	FB 90	// STD: Line and section control standard subroutines
"SYS_DPMultiDPInfo"	FB 98	FB 98	// SimpleMultiDPInfo
"SYS_DPDiagnostic"	FB 99	FB 99	// SYS: DP diagnostic and monitoring
"GCS7_StartWarning"	FB 100	FB 100	// GCS7 Start Warning Modul
"G001G_Code"	FB 101	FB 101	// Group-FB  Power supply circuit +C11
"G002G_Code"	FB 102	FB 102	// Group-FB  Contactor panel power supply 1
"G003G_Code"	FB 103	FB 103	// Group-FB  PLC monitoring
"G004G_Code"	FB 104	FB 104	// Group-FB  GENERAL ELEMENTS STEEPING
"G005G_Code"	FB 105	FB 105	// Group-FB  GENERAL ELEMENTS GERM 1
"G006G_Code"	FB 106	FB 106	// Group-FB  GENERAL ELEMENTS GERM 2
"G007G_Code"	FB 107	FB 107	// Group-FB  GENERAL ELEMENTS GERM 3
"G008G_Code"	FB 108	FB 108	// Group-FB  GENERAL ELEMENTS GERM 4
"G009G_Code"	FB 109	FB 109	// Group-FB  GENERAL ELEMENTS GERM 5
"G010G_Code"	FB 110	FB 110	// Group-FB  Line messages
"G011G_Code"	FB 111	FB 111	// Group-FB  MELE/WinCoS communication monitoring
"G012G_Code"	FB 112	FB 112	// Group-FB  GENERAL ELEMENTS GERM 6
"G013G_Code"	FB 113	FB 113	// Group-FB  GENERAL ELEMENTS GERM 7
"G014G_Code"	FB 114	FB 114	// Group-FB  GENERAL ELEMENTS GERM 8
"G015G_Code"	FB 115	FB 115	// Group-FB  CCOMPRESSED AIR PRESSURE STEEP 1 - 4
"G016G_Code"	FB 116	FB 116	// Group-FB  CCOMPRESSED AIR PRESSURE STEEP 5 - 8
"G017G_Code"	FB 117	FB 117	// Group-FB  CCOMPRESSED AIR PRESSURE STEEP 9 - 12
"G018G_Code"	FB 118	FB 118	// Group-FB  CCOMPRESSED AIR PRESSURE STEEP 13 - 16
"G019G_Code"	FB 119	FB 119	// Group-FB  CCOMPRESSED AIR PRESSURE STEEP 17 - 20
"G020G_Code"	FB 120	FB 120	// Group-FB  CCOMPRESSED AIR PRESSURE STEEP 21 - 24
"G021G_Code"	FB 121	FB 121	// Group-FB  GENERAL ELEMENTS KILN 1
"G022G_Code"	FB 122	FB 122	// Group-FB  GENERAL ELEMENTS KILN 2
"G023G_Code"	FB 123	FB 123	// Group-FB  GENERAL ELEMENTS KILN MALT TRANSFER
"G026G_Code"	FB 126	FB 126	// Group-FB  Alarm horns
"G029G_Code"	FB 129	FB 129	// Group-FB  Bin low levels
"G030G_Code"	FB 130	FB 130	// Group-FB  Bin high levels
"G031G_Code"	FB 131	FB 131	// Group-FB  GENERAL ELEMENTS STEEPING
"G032M_Code"	FB 132	FB 132	// Group-FB  CO2 FAN AND FESH AIR FLAP STEEPING 1
"G033M_Code"	FB 133	FB 133	// Group-FB  AERATION AIR STEEPING 1
"G034M_Code"	FB 134	FB 134	// Group-FB  CO2 FAN AND FESH AIR FLAP STEEPING 2
"G035M_Code"	FB 135	FB 135	// Group-FB  AERATION AIR STEEPING 2
"G036M_Code"	FB 136	FB 136	// Group-FB  CO2 FAN AND FESH AIR FLAP STEEPING 3
"G037M_Code"	FB 137	FB 137	// Group-FB  AERATION AIR STEEPING 3
"G038M_Code"	FB 138	FB 138	// Group-FB  CO2 FAN AND FESH AIR FLAP STEEPING 4
"G039M_Code"	FB 139	FB 139	// Group-FB  AERATION AIR STEEPING 4
"G040M_Code"	FB 140	FB 140	// Group-FB  CO2 FAN AND FESH AIR FLAP STEEPING 5
"G041M_Code"	FB 141	FB 141	// Group-FB  AERATION AIR STEEPING 5
"G042M_Code"	FB 142	FB 142	// Group-FB  CO2 FAN AND FESH AIR FLAP STEEPING 6
"G043M_Code"	FB 143	FB 143	// Group-FB  AERATION AIR STEEPING 6
"G044M_Code"	FB 144	FB 144	// Group-FB  CO2 FAN AND FESH AIR FLAP STEEPING 7
"G045M_Code"	FB 145	FB 145	// Group-FB  AERATION AIR STEEPING 7
"G046M_Code"	FB 146	FB 146	// Group-FB  CO2 FAN AND FESH AIR FLAP STEEPING 8
"G047M_Code"	FB 147	FB 147	// Group-FB  AERATION AIR STEEPING 8
"G048M_Code"	FB 148	FB 148	// Group-FB  CO2 FAN AND FESH AIR FLAP STEEPING 9
"G049M_Code"	FB 149	FB 149	// Group-FB  AERATION AIR STEEPING 9
"G050M_Code"	FB 150	FB 150	// Group-FB  CO2 FAN AND FESH AIR FLAP STEEPING 10
"G051M_Code"	FB 151	FB 151	// Group-FB  AERATION AIR STEEPING 10
"G052M_Code"	FB 152	FB 152	// Group-FB  CO2 FAN AND FESH AIR FLAP STEEPING 11
"G053M_Code"	FB 153	FB 153	// Group-FB  AERATION AIR STEEPING 11
"G054M_Code"	FB 154	FB 154	// Group-FB  CO2 FAN AND FESH AIR FLAP STEEPING 12
"G055M_Code"	FB 155	FB 155	// Group-FB  AERATION AIR STEEPING 12
"G056M_Code"	FB 156	FB 156	// Group-FB  CO2 FAN AND FESH AIR FLAP STEEPING 13
"G057M_Code"	FB 157	FB 157	// Group-FB  AERATION AIR STEEPING 13
"G058M_Code"	FB 158	FB 158	// Group-FB  CO2 FAN AND FESH AIR FLAP STEEPING 14
"G059M_Code"	FB 159	FB 159	// Group-FB  AERATION AIR STEEPING 14
"G060M_Code"	FB 160	FB 160	// Group-FB  CO2 FAN AND FESH AIR FLAP STEEPING 15
"G061M_Code"	FB 161	FB 161	// Group-FB  AERATION AIR STEEPING 15
"G062M_Code"	FB 162	FB 162	// Group-FB  CO2 FAN AND FESH AIR FLAP STEEPING 16
"G063M_Code"	FB 163	FB 163	// Group-FB  AERATION AIR STEEPING 16
"G064M_Code"	FB 164	FB 164	// Group-FB  CO2 FAN AND FESH AIR FLAP STEEPING 17
"G065M_Code"	FB 165	FB 165	// Group-FB  AERATION AIR STEEPING 17
"G066M_Code"	FB 166	FB 166	// Group-FB  PRODUCT SLIDER STEEPING 17
"G067M_Code"	FB 167	FB 167	// Group-FB  CO2 FAN AND FESH AIR FLAP STEEPING 18
"G068M_Code"	FB 168	FB 168	// Group-FB  AERATION AIR STEEPING 18
"G069M_Code"	FB 169	FB 169	// Group-FB  PRODUCT SLIDER STEEPING 18
"G070M_Code"	FB 170	FB 170	// Group-FB  CO2 FAN AND FESH AIR FLAP STEEPING 19
"G071M_Code"	FB 171	FB 171	// Group-FB  AERATION AIR STEEPING 19
"G072M_Code"	FB 172	FB 172	// Group-FB  PRODUCT SLIDER STEEPING 19
"G073M_Code"	FB 173	FB 173	// Group-FB  CO2 FAN AND FESH AIR FLAP STEEPING 20
"G074M_Code"	FB 174	FB 174	// Group-FB  AERATION AIR STEEPING 20
"G075M_Code"	FB 175	FB 175	// Group-FB  PRODUCT SLIDER STEEPING 20
"G076M_Code"	FB 176	FB 176	// Group-FB  CO2 FAN AND FESH AIR FLAP STEEPING 21
"G077M_Code"	FB 177	FB 177	// Group-FB  AERATION AIR STEEPING 21
"G078M_Code"	FB 178	FB 178	// Group-FB  PRODUCT SLIDER STEEPING 21
"G079M_Code"	FB 179	FB 179	// Group-FB  CO2 FAN AND FESH AIR FLAP STEEPING 22
"G080M_Code"	FB 180	FB 180	// Group-FB  AERATION AIR STEEPING 22
"G081M_Code"	FB 181	FB 181	// Group-FB  PRODUCT SLIDER STEEPING 22
"G082M_Code"	FB 182	FB 182	// Group-FB  CO2 FAN AND FESH AIR FLAP STEEPING 23
"G083M_Code"	FB 183	FB 183	// Group-FB  AERATION AIR STEEPING 23
"G084M_Code"	FB 184	FB 184	// Group-FB  PRODUCT SLIDER STEEPING 23
"G085M_Code"	FB 185	FB 185	// Group-FB  CO2 FAN AND FESH AIR FLAP STEEPING 24
"G086M_Code"	FB 186	FB 186	// Group-FB  AERATION AIR STEEPING 24
"G087M_Code"	FB 187	FB 187	// Group-FB  PRODUCT SLIDER STEEPING 24
"G090G_Code"	FB 190	FB 190	// Group-FB  GENERAL ELEMENTS GERM 1
"G091M_Code"	FB 191	FB 191	// Group-FB  BELT CONVEYOR 4100 GERM 1-4
"G092M_Code"	FB 192	FB 192	// Group-FB  BELT CONVEYOR 4200 GERM 5-8
"G093M_Code"	FB 193	FB 193	// Group-FB  BELT CONVEYOR 4300 GERM
"G094M_Code"	FB 194	FB 194	// Group-FB  BELT CONVEYOR 4400 GERM
"G095M_Code"	FB 195	FB 195	// Group-FB  BELT CONVEYOR 4500 GERM
"G097M_Code"	FB 197	FB 197	// Group-FB  LIFTING DEVICE GERM 1
"G098M_Code"	FB 198	FB 198	// Group-FB  COUPLING DEVICE TURNER GERM 1
"G099M_Code"	FB 199	FB 199	// Group-FB  COUPLING DEVICE WALL GERM 1
"G100M_Code"	FB 200	FB 200	// Group-FB  TRAVELLING DRIVE GERM 1
"G101M_Code"	FB 201	FB 201	// Group-FB  HORIZONTAL AND LIFTING SCREW GERM 1
"G102M_Code"	FB 202	FB 202	// Group-FB  LOCAL COMMAND BUTTON / LAMPS GERM 1
"G103M_Code"	FB 203	FB 203	// Group-FB  TEMPERATURE MES. GERM 1
"G104M_Code"	FB 204	FB 204	// Group-FB  TURNING SCREWS GERM 1
"G105M_Code"	FB 205	FB 205	// Group-FB  FAN AND VALVE SRAY AIR GERM 1
"G106M_Code"	FB 206	FB 206	// Group-FB  FRESH AIR LOUVER GERM 1
"G107M_Code"	FB 207	FB 207	// Group-FB  EXHAUST AIR LOUVER GERM 1
"G108M_Code"	FB 208	FB 208	// Group-FB  PRODUCT MOISTERING  GERM 1
"G109M_Code"	FB 209	FB 209	// Group-FB  HP CLEANING GERM 1
"G110M_Code"	FB 210	FB 210	// Group-FB  INLET SLIDE GERM 1
"G111M_Code"	FB 211	FB 211	// Group-FB  LOADING CONVEYOR 4600 GERM 1
"G112M_Code"	FB 212	FB 212	// Group-FB  COOLING / HEATING GERM 1
"G113M_Code"	FB 213	FB 213	// Group-FB  BELT CONVEYOR 7050 GERM 1 / 2
"G114M_Code"	FB 214	FB 214	// Group-FB  CHAIN CONVEYOR 7100 GERM
"G120G_Code"	FB 220	FB 220	// Group-FB  GENERAL ELEMENTS GERM 2
"G121M_Code"	FB 221	FB 221	// Group-FB  CHAIN CONVEYOR 4600 GERM 2
"G122M_Code"	FB 222	FB 222	// Group-FB  LIFTING DEVICE GERM 2
"G123M_Code"	FB 223	FB 223	// Group-FB  COUPLING DEVICE TURNER GERM 2
"G124M_Code"	FB 224	FB 224	// Group-FB  COUPLING DEVICE WALL GERM 2
"G125M_Code"	FB 225	FB 225	// Group-FB  TRAVELLING DRIVE GERM 2
"G126M_Code"	FB 226	FB 226	// Group-FB  HORIZONTAL AND LIFTING SCREW GERM 2
"G127M_Code"	FB 227	FB 227	// Group-FB  LOCAL COMMAND BUTTON / LAMPS GERM 2
"G128M_Code"	FB 228	FB 228	// Group-FB  TEMPERATURE MES. GERM 2
"G129M_Code"	FB 229	FB 229	// Group-FB  TURNING SCREWS GERM 2
"G130M_Code"	FB 230	FB 230	// Group-FB  FAN AND VALVE SRAY AIR GERM 2
"G131M_Code"	FB 231	FB 231	// Group-FB  FRESH AIR LOUVER GERM 2
"G132M_Code"	FB 232	FB 232	// Group-FB  EXHAUST AIR  LOUVER GERM 2
"G133M_Code"	FB 233	FB 233	// Group-FB  PRODUCT MOISTERING  GERM 2
"G134M_Code"	FB 234	FB 234	// Group-FB  HP CLEANING GERM 2
"G135M_Code"	FB 235	FB 235	// Group-FB  INLET SLIDE GERM 2
"G136M_Code"	FB 236	FB 236	// Group-FB  LOAD / UNLOAD CONVEYOR GERM 2
"G137M_Code"	FB 237	FB 237	// Group-FB  COOLING / HEATING GERM 2
"G140G_Code"	FB 240	FB 240	// Group-FB  GENERAL ELEMENTS GERM 3
"G141M_Code"	FB 241	FB 241	// Group-FB  CHAIN CONVEYOR 4600 GERM 3
"G142M_Code"	FB 242	FB 242	// Group-FB  LIFTING DEVICE GERM 3
"G143M_Code"	FB 243	FB 243	// Group-FB  COUPLING DEVICE TURNER GERM 3
"G144M_Code"	FB 244	FB 244	// Group-FB  COUPLING DEVICE WALL GERM 3
"G145M_Code"	FB 245	FB 245	// Group-FB  TRAVELLING DRIVE GERM 3
"G146M_Code"	FB 246	FB 246	// Group-FB  HORIZONTAL AND LIFTING SCREW GERM 3
"G147M_Code"	FB 247	FB 247	// Group-FB  LOCAL COMMAND BUTTON / LAMPS GERM 3
"G148M_Code"	FB 248	FB 248	// Group-FB  TEMPERATURE MES. GERM 3
"G149M_Code"	FB 249	FB 249	// Group-FB  TURNING SCREWS GERM 3
"G150M_Code"	FB 250	FB 250	// Group-FB  FAN AND VALVE SRAY AIR GERM 3
"G151M_Code"	FB 251	FB 251	// Group-FB  FRESH AIR LOUVER GERM 3
"G152M_Code"	FB 252	FB 252	// Group-FB  EXHAUST AIR LOUVER GERM 3
"G153M_Code"	FB 253	FB 253	// Group-FB  PRODUCT MOISTERING  GERM 3
"G154M_Code"	FB 254	FB 254	// Group-FB  HP CLEANING GERM 3
"G155M_Code"	FB 255	FB 255	// Group-FB  INLET SLIDE GERM 3
"G156M_Code"	FB 256	FB 256	// Group-FB  LOAD / UNLOAD CONVEYOR GERM 3
"G157M_Code"	FB 257	FB 257	// Group-FB  COOLING / HEATING GERM 3
"G158M_Code"	FB 258	FB 258	// Group-FB  CHAIN CONVEYOR 7050 GERM 3 / 4
"G160G_Code"	FB 260	FB 260	// Group-FB  GENERAL ELEMENTS GERM 4
"G161M_Code"	FB 261	FB 261	// Group-FB  CHAIN CONVEYOR 4600 GERM 4
"G162M_Code"	FB 262	FB 262	// Group-FB  LIFTING DEVICE GERM 4
"G163M_Code"	FB 263	FB 263	// Group-FB  COUPLING DEVICE TURNER GERM 4
"G164M_Code"	FB 264	FB 264	// Group-FB  COUPLING DEVICE WALL GERM 4
"G165M_Code"	FB 265	FB 265	// Group-FB  TRAVELLING DRIVE GERM 4
"G166M_Code"	FB 266	FB 266	// Group-FB  HORIZONTAL AND LIFTING SCREW GERM 4
"G167M_Code"	FB 267	FB 267	// Group-FB  LOCAL COMMAND BUTTON / LAMPS GERM 4
"G168M_Code"	FB 268	FB 268	// Group-FB  TEMPERATURE MES. GERM 4
"G169M_Code"	FB 269	FB 269	// Group-FB  TURNING SCREWS GERM 4
"G170M_Code"	FB 270	FB 270	// Group-FB  FAN AND VALVE SRAY AIR GERM 4
"G171M_Code"	FB 271	FB 271	// Group-FB  FRESH AIR LOUVER GERM 4
"G172M_Code"	FB 272	FB 272	// Group-FB  EXHAUST AIR LOUVER GERM 4
"G173M_Code"	FB 273	FB 273	// Group-FB  PRODUCT MOISTERING  GERM 4
"G174M_Code"	FB 274	FB 274	// Group-FB  HP CLEANING GERM 4
"G175M_Code"	FB 275	FB 275	// Group-FB  INLET SLIDE GERM 4
"G176M_Code"	FB 276	FB 276	// Group-FB  LOAD / UNLOAD CONVEYOR GERM 4
"G177M_Code"	FB 277	FB 277	// Group-FB  COOLING / HEATING GERM 4
"G180G_Code"	FB 280	FB 280	// Group-FB  GENERAL ELEMENTS GERM 5
"G181M_Code"	FB 281	FB 281	// Group-FB  CHAIN CONVEYOR 4600 GERM 5
"G182M_Code"	FB 282	FB 282	// Group-FB  LIFTING DEVICE GERM 5
"G183M_Code"	FB 283	FB 283	// Group-FB  COUPLING DEVICE TURNER GERM 5
"G184M_Code"	FB 284	FB 284	// Group-FB  COUPLING DEVICE WALL GERM 5
"G185M_Code"	FB 285	FB 285	// Group-FB  TRAVELLING DRIVE GERM 5
"G186M_Code"	FB 286	FB 286	// Group-FB  HORIZONTAL AND LIFTING SCREW GERM 5
"G187M_Code"	FB 287	FB 287	// Group-FB  LOCAL COMMAND BUTTON / LAMPS GERM 5
"G188M_Code"	FB 288	FB 288	// Group-FB  TEMPERATURE MES. GERM 5
"G189M_Code"	FB 289	FB 289	// Group-FB  TURNING SCREWS GERM 5
"G190M_Code"	FB 290	FB 290	// Group-FB  FAN AND VALVE SRAY AIR GERM 5
"G191M_Code"	FB 291	FB 291	// Group-FB  FRESH AIR LOUVER GERM 5
"G192M_Code"	FB 292	FB 292	// Group-FB  EXHAUST AIR LOUVER GERM 5
"G193M_Code"	FB 293	FB 293	// Group-FB  PRODUCT MOISTERING  GERM 5
"G194M_Code"	FB 294	FB 294	// Group-FB  HP CLEANING GERM 5
"G195M_Code"	FB 295	FB 295	// Group-FB  INLET SLIDE GERM 5
"G196M_Code"	FB 296	FB 296	// Group-FB  LOAD / UNLOAD CONVEYOR GERM 5
"G197M_Code"	FB 297	FB 297	// Group-FB  COOLING / HEATING GERM 5
"G198M_Code"	FB 298	FB 298	// Group-FB  CHAIN CONVEYOR 7050 GERM 5 / 6
"G200G_Code"	FB 300	FB 300	// Group-FB  GENERAL ELEMENTS GERM 6
"G201M_Code"	FB 301	FB 301	// Group-FB  CHAIN CONVEYOR 4600 GERM 6
"G202M_Code"	FB 302	FB 302	// Group-FB  LIFTING DEVICE GERM 6
"G203M_Code"	FB 303	FB 303	// Group-FB  COUPLING DEVICE TURNER GERM 6
"G204M_Code"	FB 304	FB 304	// Group-FB  COUPLING DEVICE WALL GERM 6
"G205M_Code"	FB 305	FB 305	// Group-FB  TRAVELLING DRIVE GERM 6
"G206M_Code"	FB 306	FB 306	// Group-FB  HORIZONTAL AND LIFTING SCREW GERM 6
"G207M_Code"	FB 307	FB 307	// Group-FB  LOCAL COMMAND BUTTON / LAMPS GERM 6
"G208M_Code"	FB 308	FB 308	// Group-FB  TEMPERATURE MES. GERM 6
"G209M_Code"	FB 309	FB 309	// Group-FB  TURNING SCREWS GERM 6
"G210M_Code"	FB 310	FB 310	// Group-FB  FAN AND VALVE SRAY AIR GERM 6
"G211M_Code"	FB 311	FB 311	// Group-FB  FRESH AIR LOUVER GERM 6
"G212M_Code"	FB 312	FB 312	// Group-FB  EXHAUST AIR LOUVER GERM 6
"G213M_Code"	FB 313	FB 313	// Group-FB  PRODUCT MOISTERING  GERM 6
"G214M_Code"	FB 314	FB 314	// Group-FB  HP CLEANING GERM 6
"G215M_Code"	FB 315	FB 315	// Group-FB  INLET SLIDE GERM 6
"G216M_Code"	FB 316	FB 316	// Group-FB  LOAD / UNLOAD CONVEYOR GERM 6
"G217M_Code"	FB 317	FB 317	// Group-FB  COOLING / HEATING GERM 6
"G220G_Code"	FB 320	FB 320	// Group-FB  GENERAL ELEMENTS GERM 7
"G221M_Code"	FB 321	FB 321	// Group-FB  CHAIN CONVEYOR 4600 GERM 7
"G222M_Code"	FB 322	FB 322	// Group-FB  LIFTING DEVICE GERM 7
"G223M_Code"	FB 323	FB 323	// Group-FB  COUPLING DEVICE TURNER GERM 7
"G224M_Code"	FB 324	FB 324	// Group-FB  COUPLING DEVICE WALL GERM 7
"G225M_Code"	FB 325	FB 325	// Group-FB  TRAVELLING DRIVE GERM 7
"G226M_Code"	FB 326	FB 326	// Group-FB  HORIZONTAL AND LIFTING SCREW GERM 7
"G227M_Code"	FB 327	FB 327	// Group-FB  LOCAL COMMAND BUTTON / LAMPS GERM 7
"G228M_Code"	FB 328	FB 328	// Group-FB  TEMPERATURE MES. GERM 7
"G229M_Code"	FB 329	FB 329	// Group-FB  TURNING SCREWS GERM 7
"G230M_Code"	FB 330	FB 330	// Group-FB  FAN AND VALVE SRAY AIR GERM 7
"G231M_Code"	FB 331	FB 331	// Group-FB  FRESH AIR LOUVER GERM 7
"G232M_Code"	FB 332	FB 332	// Group-FB  EXHAUST AIR LOUVER GERM 7
"G233M_Code"	FB 333	FB 333	// Group-FB  PRODUCT MOISTERING  GERM 7
"G234M_Code"	FB 334	FB 334	// Group-FB  HP CLEANING GERM 7
"G235M_Code"	FB 335	FB 335	// Group-FB  INLET SLIDE GERM 7
"G236M_Code"	FB 336	FB 336	// Group-FB  LOAD / UNLOAD CONVEYOR GERM 7
"G237M_Code"	FB 337	FB 337	// Group-FB  COOLING / HEATING GERM 7
"G238M_Code"	FB 338	FB 338	// Group-FB  CHAIN CONVEYOR 7050 GERM 7 / 8
"G240G_Code"	FB 340	FB 340	// Group-FB  GENERAL ELEMENTS GERM 8
"G241M_Code"	FB 341	FB 341	// Group-FB  CHAIN CONVEYOR 4600 GERM 8
"G242M_Code"	FB 342	FB 342	// Group-FB  LIFTING DEVICE GERM 8
"G243M_Code"	FB 343	FB 343	// Group-FB  COUPLING DEVICE TURNER GERM 8
"G244M_Code"	FB 344	FB 344	// Group-FB  COUPLING DEVICE WALL GERM 8
"G245M_Code"	FB 345	FB 345	// Group-FB  TRAVELLING DRIVE GERM 8
"G246M_Code"	FB 346	FB 346	// Group-FB  HORIZONTAL AND LIFTING SCREW GERM 8
"G247M_Code"	FB 347	FB 347	// Group-FB  LOCAL COMMAND BUTTON / LAMPS GERM 8
"G248M_Code"	FB 348	FB 348	// Group-FB  TEMPERATURE MES. GERM 8
"G249M_Code"	FB 349	FB 349	// Group-FB  TURNING SCREWS GERM 8
"G250M_Code"	FB 350	FB 350	// Group-FB  FAN AND VALVE SRAY AIR GERM 8
"G251M_Code"	FB 351	FB 351	// Group-FB  FRESH AIR LOUVER GERM 8
"G252M_Code"	FB 352	FB 352	// Group-FB  EXHAUST AIR LOUVER GERM 8
"G253M_Code"	FB 353	FB 353	// Group-FB  PRODUCT MOISTERING  GERM 8
"G254M_Code"	FB 354	FB 354	// Group-FB  HP CLEANING GERM 8
"G255M_Code"	FB 355	FB 355	// Group-FB  INLET SLIDE GERM 8
"G256M_Code"	FB 356	FB 356	// Group-FB  LOAD / UNLOAD CONVEYOR GERM 8
"G257M_Code"	FB 357	FB 357	// Group-FB  COOLING / HEATING GERM 8
"G260G_Code"	FB 360	FB 360	// Group-FB  GENERAL ELEMENTS KILN 1
"G261M_Code"	FB 361	FB 361	// Group-FB  BELT CONVEYOR 7200 KILN
"G262M_Code"	FB 362	FB 362	// Group-FB  BELT CONVEYOR 7300 KILN
"G263M_Code"	FB 363	FB 363	// Group-FB  BELT CONVEYOR 7301 KILN
"G264M_Code"	FB 364	FB 364	// Group-FB  BELT CONVEYOR 7400 KILN
"G265M_Code"	FB 365	FB 365	// Group-FB  LIFTING DEVICE KILN 1
"G266M_Code"	FB 366	FB 366	// Group-FB  TRAVELLING DRIVE KILN 1
"G267M_Code"	FB 367	FB 367	// Group-FB  UNLOADING / LOADING SCREW KILN 1
"G268M_Code"	FB 368	FB 368	// Group-FB  DISCHARGE DOOR KILN 1
"G269M_Code"	FB 369	FB 369	// Group-FB  TEMPERATURE MES. KILN 1
"G270M_Code"	FB 370	FB 370	// Group-FB  AIR SHUT SLIDE KILN 1
"G271M_Code"	FB 371	FB 371	// Group-FB  FAN KILN 1
"G272M_Code"	FB 372	FB 372	// Group-FB  FRESH AIR RECYCLING KILN 1
"G273M_Code"	FB 373	FB 373	// Group-FB  RECYCLING AIR LOUVER KILN 1
"G274M_Code"	FB 374	FB 374	// Group-FB  EXHAUST AIR LOUVER KILN 1
"G275M_Code"	FB 375	FB 375	// Group-FB  BYPASS FLAP KILN 1
"G276M_Code"	FB 376	FB 376	// Group-FB  HEATING KILN 1
"G277M_Code"	FB 377	FB 377	// Group-FB  LOUVER AIR HEATER KILN 1
"G278M_Code"	FB 378	FB 378	// Group-FB  WITHERING AIR KILN 1
"G279M_Code"	FB 379	FB 379	// Group-FB  HEATING KILN 1 + 2
"G280M_Code"	FB 380	FB 380	// Group-FB  CHAIN CONVEYOR 9001 KILN 1
"G281M_Code"	FB 381	FB 381	// Group-FB  ELEVATOR 9002 AFTER KILN
"G282M_Code"	FB 382	FB 382	// Group-FB  FLAP BOX 9008
"G283M_Code"	FB 383	FB 383	// Group-FB  CULM BATCH BIN 9005
"G284M_Code"	FB 384	FB 384	// Group-FB  BELT CONVEYOR 7100 KILN
"G290G_Code"	FB 390	FB 390	// Group-FB  GENERAL ELEMENTS KILN 2
"G291M_Code"	FB 391	FB 391	// Group-FB  LIFTING DEVICE KILN 2
"G292M_Code"	FB 392	FB 392	// Group-FB  TRAVELLING DRIVE KILN 2
"G293M_Code"	FB 393	FB 393	// Group-FB  UNLOADING / LOADING SCREW KILN 2
"G294M_Code"	FB 394	FB 394	// Group-FB  DISCHARGE DOOR KILN 2
"G295M_Code"	FB 395	FB 395	// Group-FB  TEMPERATURE MES. KILN 2
"G296M_Code"	FB 396	FB 396	// Group-FB  AIR SHUT SLIDE KILN 2
"G297M_Code"	FB 397	FB 397	// Group-FB  FAN KILN 2
"G298M_Code"	FB 398	FB 398	// Group-FB  FRESH AIR FLAP KILN 2
"G299M_Code"	FB 399	FB 399	// Group-FB  RECYCLING AIR FLAP KILN 2
"G300M_Code"	FB 400	FB 400	// Group-FB  EXHAUST AIR FLAP KILN 2
"G301M_Code"	FB 401	FB 401	// Group-FB  BYPASS FLAP KILN 2
"G302M_Code"	FB 402	FB 402	// Group-FB  HEATING KILN 2
"G303M_Code"	FB 403	FB 403	// Group-FB  LOUVER AIR HEATER KILN 2
"G304M_Code"	FB 404	FB 404	// Group-FB  WITHERING AIR KILN 2
"G305M_Code"	FB 405	FB 405	// Group-FB  CHAIN CONVEYOR 9002 KILN 2
"G306M_Code"	FB 406	FB 406	// Group-FB  DMBG DISCHARGER KILN MALT TRANSFER
"G307M_Code"	FB 407	FB 407	// Group-FB  SCREW CONVEYOR 9007 KILN MALT TRANSFER
"G308M_Code"	FB 408	FB 408	// Group-FB  BELT CONVEYOR 9009 KILN MALT TRANSFER
"G309M_Code"	FB 409	FB 409	// Group-FB  ELEVATOR EXCISTING
"G310M_Code"	FB 410	FB 410	// Group-FB  PLC1 TO EXCISTING DEGERMINATION SYSTEM
"G311M_Code"	FB 411	FB 411	// Group-FB  CENTRAL ASPIRATION UNLOAD KILN
"G320M_Code"	FB 420	FB 420	// Group-FB  PCC GRAPHIC SUPPORT
"SSA_MH_EventsToPIC"	FB 470	FB 470
"SSA_MH_Step_Values"	FB 472	FB 472	// Malthaouse. Log Step Values
"STD_StartupBinTime"	FB 801	FB 801	// STD: Startup bin filling procedure
"SSA_PneumaticControl_Fct"	FB 841	FB 841	// SSA: Pneumatic controller
"SSW_EL_ASI_Fct"	FB 899	FB 899	// Element Control ASI Master Wago/Profibus
"A_1911_MXZ0MA_Code"	FB 1000	FB 1000	// Machine-FB (FB50) BELT CONVEYOR 4100 GERM 1-4
"A_1915_MXZ01MA_Code"	FB 1001	FB 1001	// Machine-FB (FB50) BELT CONVEYOR 4200 GERM 5-8
"A_1921_MXZ01MA_Code"	FB 1002	FB 1002	// Machine-FB (FB50) BELT CONVEYOR 4300
"A_1931_MXZ0MA_Code"	FB 1003	FB 1003	// Machine-FB (FB50) BELT CONVEYOR 4400
"A_1941_MXZ01MA_Code"	FB 1004	FB 1004	// Machine-FB (FB50) BELT CONVEYOR 4500
"A_1942_MXZ0MA_Code"	FB 1005	FB 1005	// Machine-FB (FB50) CHUTE DRIVE
"A_2111_MXZ41MA_Code"	FB 1006	FB 1006	// Machine-FB (FB86) TRAVELING DRIVE
"A_2115_MXZ11MA_Code"	FB 1007	FB 1007	// Machine-FB (FB50) HORIZONTAL SCREW
"A_2115_MXZ15MA_Code"	FB 1008	FB 1008	// Machine-FB (FB50) LIFTING SCREW
"A_2101_MXZ01MA_Code"	FB 1009	FB 1009	// Machine-FB (FB50) BELT CONVEYOR 4600
"A_2911_MXZ01MA_Code"	FB 1010	FB 1010	// Machine-FB (FB50) BELT CONVEYOR 4600 GERM 1
"A_2926_MXZ0MA_Code"	FB 1011	FB 1011	// Machine-FB (FB50) BELT CONVEYOR 7200
"A_2929_MXZ0MA_Code"	FB 1012	FB 1012	// Machine-FB (FB50) BELT CONVEYOR 7300
"A_2932_MXZ0MA1_Code"	FB 1013	FB 1013	// Machine-FB (FB50) BELT CONVEYOR 7301 MA1
"A_2932_MXZ0MA2_Code"	FB 1014	FB 1014	// Machine-FB (FB50) BELT CONVEYOR 7301 MA2
"A_2935_MXZ01MA_Code"	FB 1015	FB 1015	// Machine-FB (FB50) BELT CONVEYOR 7400
"A_3111_MXZ21_31MA_Code"	FB 1016	FB 1016	// Machine-FB (FB85) LIFTING DRIVE
"A_3111_MXZ41MA_Code"	FB 1017	FB 1017	// Machine-FB (FB86) TRAVELING DRIVE
"A_3125_MXZ01MA_Code"	FB 1018	FB 1018	// Machine-FB (FB50) FAN 1
"A_3126_MXZ01MA_Code"	FB 1019	FB 1019	// Machine-FB (FB50) FAN 2
"A_3921_MXZ01MA_Code"	FB 1020	FB 1020	// Machine-FB (FB50) CHAIN CONVEYOR UNDER KILN 1
"A_3924_MXZ01MA_Code"	FB 1021	FB 1021	// Machine-FB (FB60) ASPIRATION UNDER KILN 1
"A_3930_MXZ01MA_Code"	FB 1022	FB 1022	// Machine-FB (FB50) ELEVATOR
"A_3932_MXZ01MA_Code"	FB 1023	FB 1023	// Machine-FB (FB60) FILTER ASPIRATION ELEVATOR
"A_2923_MXZ0MA_Code"	FB 1024	FB 1024	// Machine-FB (FB50) BELT CONVEYOR 7100
"A_3914_MXZ01MA_Code"	FB 1025	FB 1025	// Machine-FB (FB60) ASPIRATION UNDER KILN 2
"A_3911_MXZ01MA_Code"	FB 1026	FB 1026	// Machine-FB (FB50) CHAIN CONVEYOR UNDER KILN 2
"A_3955_MXZ01MA_Code"	FB 1027	FB 1027	// Machine-FB (FB50) SCREW CONVEYOR DRIVE
"A_3938_MXZ01MA_Code"	FB 1028	FB 1028	// Machine-FB (FB50) BELT CONVEYOR 9009
"A_3945_MXZ01MA_Code"	FB 1029	FB 1029	// Machine-FB (FB50) EXCISTING ELEVATOR
"A_3960_MXZ01MA_Code"	FB 1030	FB 1030	// Machine-FB (FB60) FAN DRIVE CENTRAL ASPIRATION
"COM_PLCSend"	FB 1701	FB 1701	// COM: Send data to an other PLC
"COM_PLCReceive"	FB 1702	FB 1702	// COM: Receive data from an other PLC
"STD_PLCWatchdog"	FB 1703	FB 1703	// STD: PLC to PLC communication watchdog
"COM_Modbus_CMV96"	FB 1709	FB 1709	// Modbus interface to CMV96
"SSA_EL_Sampler_RFID"	FB 1714	FB 1714	// Baumer RFID
"SSA_SEW_MOVIDRIVE"	FB 1812	FB 1812	// SEW MOVIDRIVE Frequency Inverter Profibus Communication
"SSA_ABB"	FB 1816	FB 1816	// ABB ACS800 Frequency Inverter Profibus Communication
"SYS_CBitCtrl"	FC 2	FC 2	// SYS: Call change bit controller
"SYS_DirectCtrl"	FC 3	FC 3	// GCS7: PC direct control subroutines
"SYS_Horn_Code"	FC 4	FC 4	// GCS7: Code Horn Modul
"AG_SEND"	FC 5	FC 5	// Send Function for SEND-/RECEIVE-Services to SIMATIC NET CPs
"AG_RECEIVE"	FC 6	FC 6	// Receive Function for SEND-/RECEIVE-Services to SIMATIC NET CPs
"SYS_CallGroup"	FC 9	FC 9	// SYS: Call group functions blocks
"ASW_SimulElements"	FC 10	FC 10	// USW: Element simulation
"SYS_CallLineSection"	FC 11	FC 11	// SYS: Call line and section controller
"SYS_RW_IO"	FC 12	FC 12	// SYS: Read/Write IO of elements
"TEST_IOSIMULI_Copy"	FC 16	FC 16	// TEST: Functions for serial IO-Manager
"GCS7_TON_LONG"	FC 17	FC 17	// Timer TON long time values
"GCS7_TON"	FC 18	FC 18	// Timer TON
"SYS_Analog_S5_to_S7"	FC 19	FC 19	// Convert analog value S5 format to S7 for
"CWA_ScaleSimul"	FC 39	FC 39	// CWA: Scale simulation
"CWA_ScaleCtrlSub"	FC 40	FC 40	// CWA: Scale control subroutines
"CWA_ScaleCtrlMain"	FC 41	FC 41	// CWA: Scale control main program
"CWA_ScaleRead"	FC 42	FC 42	// CWA: Scale read
"GCS7_LogConvert"	FC 45	FC 45	// LOG: GCS7 message convert
"SYS_LOG_EntryQueue"	FC 46	FC 46	// LOG: Message entry in queue
"SYS_LOG_CtrlQueue"	FC 47	FC 47	// LOG: Call queue controller
"SYS_Copy_DBtoDB"	FC 49	FC 49	// SYS: Block transfer DB to DB
"SYS_Copy_Array_Element"	FC 50	FC 50
"SYS_DeleteDB"	FC 51	FC 51	// BASIS: Delete data block
"SYS_InitFlagTimer"	FC 52	FC 52	// SYS: Init flags and timers
"SYS_BitAddress"	FC 53	FC 53	// Get Bit Adress of any Symbol
"GCS7_LineCtrlMain"	FC 58	FC 58	// GCS7: Line control main program
"GCS7_LineCtrlSub"	FC 59	FC 59	// GCS7: Line control subroutines
"GCS7_SecCtrlMain"	FC 60	FC 60	// GCS7: Section control main program
"GCS7_SecCtrlSub"	FC 61	FC 61	// GCS7: Section control subroutines
"GCS7_SecCtrlASW"	FC 63	FC 63	// GCS7: Section control ASW subroutines
"GCS7_BinCtrlMain"	FC 66	FC 66	// GCS7: Bin control main program
"GCS7_BinCtrlSub"	FC 67	FC 67	// GCS7: Scale control subroutines
"GCS7_ScaleCtrlMain"	FC 68	FC 68	// GCS7: Scale control main program
"GCS7_ScaleCtrlSub"	FC 69	FC 69	// GCS7: Scale control subroutines
"GCS7_LogConvert_10"	FC 73	FC 73	// LOG: GCS7 message convert Format 10
"SYS_DPDiagMain"	FC 75	FC 75	// DPDiagnose Main program
"SYS_DPDiag1"	FC 76	FC 76	// DPDiagnose => not Siemens Slave
"GCS7BinCtrlUpdataLevel"	FC 78	FC 78	// GCS7: Bin Control Update Bin Level
"ASW_GraphicFunction"	FC 80	FC 80
"ASW_PlantParFunction"	FC 81	FC 81
"SIEMENS_IECFC6_DT_DATE"	FC 90	FC 90	// SIEMENS: Date from DATE_AND_TIME
"SIEMENS_IECFC8_DT_TOD"	FC 91	FC 91	// SIEMENS: Time from DATE_AND_TIME
"SIEMENS_IECFC3_D_TOD_DT"	FC 92	FC 92	// SIEMENS: DATE+TIME_OF_DAY --> DATE_AND_TIME
"SIEMENS_IECFC10_EQ_STR"	FC 93	FC 93	// SIEMENS: String Compare
"SYS_SimpleDPInfo"	FC 98	FC 98	// SYS: PROFIBUS-DP diagnostic
"SIEMENS_GlobalDPInfo"	FC 99	FC 99	// SIEMENS: PROFIBUS-DP monitoring
"SYS_GeneralPLCStartup"	FC 100	FC 100	// SYS: General plc startup functions
"SYS_GeneralFunctions"	FC 105	FC 105	// SYS: General plant signals
"HW_PanelLamps"	FC 106	FC 106	// HW: Lamps on control panel
"ConvertGrayCode"	FC 108	FC 108	// Convert Gray Code
"SSA_Analog_S5_to_S7"	FC 109	FC 109	// Convert analog value S5 format to S7 for
"TEST_Functions"	FC 111	FC 111	// TEST: Testfunctions
"STD_LineSecStdSub"	FC 120	FC 120	// STD: Line and section control standard subroutines
"STD_OnOffSignals"	FC 121	FC 121	// STD: ON / OFF Signal handling
"STD_OnOffSignals32"	FC 122	FC 122	// STD: ON / OFF Signal handling with 32-Bit
"COM_PLCtoPLC"	FC 141	FC 141	// COM: PLC to PLC communication
"VDU_MsgQueueEntry"	FC 145	FC 145	// VDU: Message entry into queue
"USW_CWAFastOperations"	FC 151	FC 151	// USW: Fast CWA operation, called by interrupt ob
"STD_SearchChangeBit"	FC 241	FC 241	// STD: Search object change bits
"STD_PLCLiveValue"	FC 242	FC 242	// STD: Live value handling for PCC
"STD_MinMaxSearch"	FC 243	FC 243	// STD: Search for min/max values
"STD_AuxiliaryFunctions"	FC 247	FC 247	// STD: Auxiliary functions
"STD_EdgeFunctions"	FC 248	FC 248	// STD: Edge / step functions
"STD_ScaleAnalogSignal"	FC 249	FC 249	// STD: Convert SIEMENS S5 analog values
"STD_QueueManager"	FC 251	FC 251	// STD: Queue manager main program
"STD_QueueSub"	FC 252	FC 252	// STD: Queue manager sub program copy/search
"STD_QueueIdx"	FC 253	FC 253	// STD: Queue manager sub program index
"STD_QueueFilter"	FC 254	FC 254	// STD: Queue manager sub program compare
"STD_QueueModEntry"	FC 256	FC 256	// STD: Queue manager log queue entry
"ASW_MAL1Ctrl"	FC 800	FC 800	// ASW: Line functions
"ASW_MAL1S001Ctrl"	FC 801	FC 801	// ASW: Section functions
"ASW_MAL1S005Ctrl"	FC 805	FC 805	// ASW: Section functions
"ASW_MAL1S006Ctrl"	FC 806	FC 806	// ASW: Section functions
"ASW_MAL1S007Ctrl"	FC 807	FC 807	// ASW: Section functions
"ASW_MAL1S017Ctrl"	FC 817	FC 817	// ASW: Section functions
"ASW_MAL1S018Ctrl"	FC 818	FC 818	// ASW: Section functions
"ASW_MAL1S019Ctrl"	FC 819	FC 819	// ASW: Section functions
"ASW_MAL1S020Ctrl"	FC 820	FC 820	// ASW: Section functions
"ASW_MAL1S021Ctrl"	FC 821	FC 821	// ASW: Section functions
"ASW_MAL1S022Ctrl"	FC 822	FC 822	// ASW: Section functions
"ASW_MAL1S023Ctrl"	FC 823	FC 823	// ASW: Section functions
"ASW_MAL1S024Ctrl"	FC 824	FC 824	// ASW: Section functions
"ASW_MAL1S032Ctrl"	FC 832	FC 832	// ASW: Section functions
"ASW_MAL1S033Ctrl"	FC 833	FC 833	// ASW: Section functions
"ASW_MAL1S034Ctrl"	FC 834	FC 834	// ASW: Section functions
"Act_Value_LogConvert"	FC 1045	FC 1045	// LOG: GCS7 message convert
"SSA_MH_LogEntry_ActValue"	FC 1046	FC 1046	// LOG: Message entry in queue
"SSA_MH_LogCtrl_ActValue"	FC 1047	FC 1047	// LOG: Call queue controller
"SSA_MH_Increment_counter"	FC 1048	FC 1048
"Takt/Pause"	FC 1105	FC 1105
"Takt mit Pause"	FC 1106	FC 1106	// Takt/Pause AWR
"ASW_StageCtrl_Fct"	FC 1800	FC 1800
"SIEMENS_IEC_D_TOD_DT"	FC 2003	FC 2003	// SIEMENS: DATE+TIME_OF_DAY --> DATE_AND_TIME
"SSA_Vis_Update"	FC 2042	FC 2042	// Update Handshake for Graphik Update
"SSA_VIS_Status"	FC 2043	FC 2043	// Convert Status for Viscontrol
"SSA_VIS_Log_Msg"	FC 2055	FC 2055	// Enter Viscontrol Log Message
"A_11_A040Z1_I1"	I 12.0	BOOL	// POWER SUPPLY FAILURE +C11
"A_11_S_H097Z1_I1"	I 12.1	BOOL	// OPERATING ON +C11
"A_11_K091Z1_I1"	I 12.2	BOOL	// FUSE SWITCH OFF +C11
"A_11_A097Z1_I1"	I 12.3	BOOL	// EMERGENCY-STOP +C11
"A_11_F043Z1_I1"	I 12.4	BOOL	// POWER SUPPLY HEATING +C11
"A_1199_SHE01_I1"	I 13.0	BOOL	// EMERGENCY-OFF STEEPING HOUSE +25m
"A_1199_SHE02_I1"	I 13.1	BOOL	// EMERGENCY-OFF STEEPING HOUSE +35m
"A_1111_MXZ11_I1"	I 24.0	BOOL	// ASPIRATION FAN TANK 1
"A_1112_MXZ11_I1"	I 24.1	BOOL	// ASPIRATION FAN TANK 2
"A_1113_MXZ11_I1"	I 24.2	BOOL	// ASPIRATION FAN TANK 3
"A_1114_MXZ11_I1"	I 24.3	BOOL	// ASPIRATION FAN TANK 4
"A_1115_MXZ11_I1"	I 24.4	BOOL	// ASPIRATION FAN TANK 5
"A_1116_MXZ11_I1"	I 24.5	BOOL	// ASPIRATION FAN TANK 6
"A_1117_MXZ11_I1"	I 24.6	BOOL	// ASPIRATION FAN TANK 7
"A_1118_MXZ11_I1"	I 24.7	BOOL	// ASPIRATION FAN TANK 8
"A_1119_MXZ11_I1"	I 25.0	BOOL	// ASPIRATION FAN TANK 9
"A_1120_MXZ11_I1"	I 25.1	BOOL	// ASPIRATION FAN TANK 10
"A_1121_MXZ11_I1"	I 25.2	BOOL	// ASPIRATION FAN TANK 11
"A_1122_MXZ11_I1"	I 25.3	BOOL	// ASPIRATION FAN TANK 12
"A_1123_MXZ11_I1"	I 25.4	BOOL	// ASPIRATION FAN TANK 13
"A_1124_MXZ11_I1"	I 25.5	BOOL	// ASPIRATION FAN TANK 14
"A_1125_MXZ11_I1"	I 25.6	BOOL	// ASPIRATION FAN TANK 15
"A_1126_MXZ11_I1"	I 25.7	BOOL	// ASPIRATION FAN TANK 16
"A_1127_MXZ11_I1"	I 26.0	BOOL	// ASPIRATION FAN TANK 17
"A_1127_MXZ21_I1"	I 26.1	BOOL	// DISCHARGE SLIDE T17 CLOSED
"A_1127_MXZ21_I2"	I 26.2	BOOL	// DISCHARGE SLIDE T17 OPENED
"A_1128_MXZ11_I1"	I 26.3	BOOL	// ASPIRATION FAN TANK 18
"A_1128_MXZ21_I1"	I 26.4	BOOL	// DISCHARGE SLIDE T18 CLOSED
"A_1128_MXZ21_I2"	I 26.5	BOOL	// DISCHARGE SLIDE T18 OPENED
"A_1129_MXZ11_I1"	I 26.6	BOOL	// ASPIRATION FAN TANK 19
"A_1129_MXZ21_I1"	I 26.7	BOOL	// DISCHARGE SLIDE T19 CLOSED
"A_1129_MXZ21_I2"	I 27.0	BOOL	// DISCHARGE SLIDE T19 OPENED
"A_1130_MXZ11_I1"	I 27.1	BOOL	// ASPIRATION FAN TANK 20
"A_1130_MXZ21_I1"	I 27.2	BOOL	// DISCHARGE SLIDE T20 CLOSED
"A_1130_MXZ21_I2"	I 27.3	BOOL	// DISCHARGE SLIDE T20 OPENED
"A_1131_MXZ11_I1"	I 27.4	BOOL	// ASPIRATION FAN TANK 21
"A_1131_MXZ21_I1"	I 27.5	BOOL	// DISCHARGE SLIDE T21 CLOSED
"A_1131_MXZ21_I2"	I 27.6	BOOL	// DISCHARGE SLIDE T21 OPENED
"A_1132_MXZ11_I1"	I 27.7	BOOL	// ASPIRATION FAN TANK 22
"A_1132_MXZ21_I1"	I 28.0	BOOL	// DISCHARGE SLIDE T22 CLOSED
"A_1132_MXZ21_I2"	I 28.1	BOOL	// DISCHARGE SLIDE T22 OPENED
"A_1133_MXZ11_I1"	I 28.2	BOOL	// ASPIRATION FAN TANK 23
"A_1133_MXZ21_I1"	I 28.3	BOOL	// DISCHARGE SLIDE T23 CLOSED
"A_1133_MXZ21_I2"	I 28.4	BOOL	// DISCHARGE SLIDE T23 OPENED
"A_1134_MXZ11_I1"	I 28.5	BOOL	// ASPIRATION FAN TANK 24
"A_1134_MXZ21_I1"	I 28.6	BOOL	// DISCHARGE SLIDE T24 CLOSED
"A_1134_MXZ21_I2"	I 28.7	BOOL	// DISCHARGE SLIDE T24 OPENED
"A_1151_MXZ11_I1"	I 29.0	BOOL	// COMPRESSED AIR GROUP S1-S4
"A_1152_MXZ11_I1"	I 29.1	BOOL	// COMPRESSED AIR GROUP S5-S8
"A_1153_MXZ11_I1"	I 29.2	BOOL	// COMPRESSED AIR GROUP S9-S12
"A_1154_MXZ11_I1"	I 29.3	BOOL	// COMPRESSED AIR GROUP S13-S16
"A_1155_MXZ11_I1"	I 29.4	BOOL	// COMPRESSED AIR GROUP S17-S20
"A_1156_MXZ11_I1"	I 29.5	BOOL	// COMPRESSED AIR GROUP S21-S24
"A_1111_BZS41_I1"	I 32.0	BOOL	// FRESH-AIR TANK 1 CLOSED
"A_1111_BZS42_I1"	I 32.1	BOOL	// FRESH-AIR TANK 1 OPENED
"A_1112_BZS41_I1"	I 32.2	BOOL	// FRESH-AIR TANK 2 CLOSED
"A_1112_BZS42_I1"	I 32.3	BOOL	// FRESH-AIR TANK 2 OPENED
"A_1113_BZS41_I1"	I 32.4	BOOL	// FRESH-AIR TANK 3 CLOSED
"A_1113_BZS42_I1"	I 32.5	BOOL	// FRESH-AIR TANK 3 OPENED
"A_1114_BZS41_I1"	I 32.6	BOOL	// FRESH-AIR TANK 4 CLOSED
"A_1114_BZS42_I1"	I 32.7	BOOL	// FRESH-AIR TANK 4 OPENED
"A_1115_BZS41_I1"	I 33.0	BOOL	// FRESH-AIR TANK 5 CLOSED
"A_1115_BZS42_I1"	I 33.1	BOOL	// FRESH-AIR TANK 5 OPENED
"A_1116_BZS41_I1"	I 33.2	BOOL	// FRESH-AIR TANK 6 CLOSED
"A_1116_BZS42_I1"	I 33.3	BOOL	// FRESH-AIR TANK 6 OPENED
"A_1117_BZS41_I1"	I 33.4	BOOL	// FRESH-AIR TANK 7 CLOSED
"A_1117_BZS42_I1"	I 33.5	BOOL	// FRESH-AIR TANK 7 OPENED
"A_1118_BZS41_I1"	I 33.6	BOOL	// FRESH-AIR TANK 8 CLOSED
"A_1118_BZS42_I1"	I 33.7	BOOL	// FRESH-AIR TANK 8 OPENED
"A_1119_BZS41_I1"	I 34.0	BOOL	// FRESH-AIR TANK 9 CLOSED
"A_1119_BZS42_I1"	I 34.1	BOOL	// FRESH-AIR TANK 9 OPENED
"A_1120_BZS41_I1"	I 34.2	BOOL	// FRESH-AIR TANK 10 CLOSED
"A_1120_BZS42_I1"	I 34.3	BOOL	// FRESH-AIR TANK 10 OPENED
"A_1121_BZS41_I1"	I 34.4	BOOL	// FRESH-AIR TANK 11 CLOSED
"A_1121_BZS42_I1"	I 34.5	BOOL	// FRESH-AIR TANK 11 OPENED
"A_1122_BZS41_I1"	I 34.6	BOOL	// FRESH-AIR TANK 12 CLOSED
"A_1122_BZS42_I1"	I 34.7	BOOL	// FRESH-AIR TANK 12 OPENED
"A_1123_BZS41_I1"	I 44.0	BOOL	// FRESH-AIR TANK 13 CLOSED
"A_1123_BZS42_I1"	I 44.1	BOOL	// FRESH-AIR TANK 13 OPENED
"A_1124_BZS41_I1"	I 44.2	BOOL	// FRESH-AIR TANK 14 CLOSED
"A_1124_BZS42_I1"	I 44.3	BOOL	// FRESH-AIR TANK 14 OPENED
"A_1125_BZS41_I1"	I 44.4	BOOL	// FRESH-AIR TANK 15 CLOSED
"A_1125_BZS42_I1"	I 44.5	BOOL	// FRESH-AIR TANK 15 OPENED
"A_1126_BZS41_I1"	I 44.6	BOOL	// FRESH-AIR TANK 16 CLOSED
"A_1126_BZS42_I1"	I 44.7	BOOL	// FRESH-AIR TANK 16 OPENED
"A_1127_BZS41_I1"	I 45.0	BOOL	// FRESH-AIR TANK 17 CLOSED
"A_1127_BZS42_I1"	I 45.1	BOOL	// FRESH-AIR TANK 17 OPENED
"A_1128_BZS41_I1"	I 45.2	BOOL	// FRESH-AIR TANK 18 CLOSED
"A_1128_BZS42_I1"	I 45.3	BOOL	// FRESH-AIR TANK 18 OPENED
"A_1129_BZS41_I1"	I 45.4	BOOL	// FRESH-AIR TANK 19 CLOSED
"A_1129_BZS42_I1"	I 45.5	BOOL	// FRESH-AIR TANK 19 OPENED
"A_1130_BZS41_I1"	I 45.6	BOOL	// FRESH-AIR TANK 20 CLOSED
"A_1130_BZS42_I1"	I 45.7	BOOL	// FRESH-AIR TANK 20 OPENED
"A_1131_BZS41_I1"	I 46.0	BOOL	// FRESH-AIR TANK 21 CLOSED
"A_1131_BZS42_I1"	I 46.1	BOOL	// FRESH-AIR TANK 21 OPENED
"A_1132_BZS41_I1"	I 46.2	BOOL	// FRESH-AIR TANK 22 CLOSED
"A_1132_BZS42_I1"	I 46.3	BOOL	// FRESH-AIR TANK 22 OPENED
"A_1133_BZS41_I1"	I 46.4	BOOL	// FRESH-AIR TANK 23 CLOSED
"A_1133_BZS42_I1"	I 46.5	BOOL	// FRESH-AIR TANK 23 OPENED
"A_1134_BZS41_I1"	I 46.6	BOOL	// FRESH-AIR TANK 24 CLOSED
"A_1134_BZS42_I1"	I 46.7	BOOL	// FRESH-AIR TANK 24 OPENED
"A_1161_MXZ01_I1"	I 48.0	BOOL	// SLIDE GATE 1 - CO2 OPEN
"A_1161_MXZ01_I2"	I 48.1	BOOL	// SLIDE GATE 1 - CO2 CLOSE
"A_1161_BZS01_I1"	I 48.2	BOOL	// SLIDE GATE 1 - CO2 CLOSED
"A_1161_BZS02_I1"	I 48.3	BOOL	// SLIDE GATE 1 - CO2 OPENED
"A_1162_MXZ01_I1"	I 48.4	BOOL	// SLIDE GATE 2 - CO2 OPEN
"A_1162_MXZ01_I2"	I 48.5	BOOL	// SLIDE GATE 2 - CO2 CLOSE
"A_1162_BZS01_I1"	I 48.6	BOOL	// SLIDE GATE 2 - CO2 CLOSED
"A_1162_BZS02_I1"	I 48.7	BOOL	// SLIDE GATE 2 - CO2 OPENED
"A_1163_MXZ01_I1"	I 49.0	BOOL	// SLIDE GATE 3 - CO2 OPEN
"A_1163_MXZ01_I2"	I 49.1	BOOL	// SLIDE GATE 3 - CO2 CLOSE
"A_1163_BZS01_I1"	I 49.2	BOOL	// SLIDE GATE 3 - CO2 CLOSED
"A_1163_BZS02_I1"	I 49.3	BOOL	// SLIDE GATE 3 - CO2 OPENED
"A_1164_MXZ01_I1"	I 49.4	BOOL	// SLIDE GATE 4 - CO2 OPEN
"A_1164_MXZ01_I2"	I 49.5	BOOL	// SLIDE GATE 4 - CO2 CLOSE
"A_1164_BZS01_I1"	I 49.6	BOOL	// SLIDE GATE 4 - CO2 CLOSED
"A_1164_BZS02_I1"	I 49.7	BOOL	// SLIDE GATE 4 - CO2 OPENED
"A_1165_MXZ01_I1"	I 50.0	BOOL	// SLIDE GATE 5 - CO2 OPEN
"A_1165_MXZ01_I2"	I 50.1	BOOL	// SLIDE GATE 5 - CO2 CLOSE
"A_1165_BZS01_I1"	I 50.2	BOOL	// SLIDE GATE 5 - CO2 CLOSED
"A_1165_BZS02_I1"	I 50.3	BOOL	// SLIDE GATE 5 - CO2 OPENED
"A_1166_MXZ01_I1"	I 50.4	BOOL	// SLIDE GATE 6 - CO2 OPEN
"A_1166_MXZ01_I2"	I 50.5	BOOL	// SLIDE GATE 6 - CO2 CLOSE
"A_1166_BZS01_I1"	I 50.6	BOOL	// SLIDE GATE 6 - CO2 CLOSED
"A_1166_BZS02_I1"	I 50.7	BOOL	// SLIDE GATE 6 - CO2 OPENED
"A_1167_MXZ01_I1"	I 51.0	BOOL	// SLIDE GATE 7 - CO2 OPEN
"A_1167_MXZ01_I2"	I 51.1	BOOL	// SLIDE GATE 7 - CO2 CLOSE
"A_1167_BZS01_I1"	I 51.2	BOOL	// SLIDE GATE 7 - CO2 CLOSED
"A_1167_BZS02_I1"	I 51.3	BOOL	// SLIDE GATE 7 - CO2 OPENED
"A_1168_MXZ01_I1"	I 51.4	BOOL	// SLIDE GATE 8 - CO2 OPEN
"A_1168_MXZ01_I2"	I 51.5	BOOL	// SLIDE GATE 8 - CO2 CLOSE
"A_1168_BZS01_I1"	I 51.6	BOOL	// SLIDE GATE 8 - CO2 CLOSED
"A_1168_BZS02_I1"	I 51.7	BOOL	// SLIDE GATE 8 - CO2 OPENED
"A_1169_MXZ01_I1"	I 52.0	BOOL	// SLIDE GATE 9 - CO2 OPEN
"A_1169_MXZ01_I2"	I 52.1	BOOL	// SLIDE GATE 9 - CO2 CLOSE
"A_1169_BZS01_I1"	I 52.2	BOOL	// SLIDE GATE 9 - CO2 CLOSED
"A_1169_BZS02_I1"	I 52.3	BOOL	// SLIDE GATE 9 - CO2 OPENED
"A_1170_MXZ01_I1"	I 52.4	BOOL	// SLIDE GATE 10-CO2 OPEN
"A_1170_MXZ01_I2"	I 52.5	BOOL	// SLIDE GATE 10-CO2 CLOSE
"A_1170_BZS01_I1"	I 52.6	BOOL	// SLIDE GATE 10-CO2 CLOSED
"A_1170_BZS02_I1"	I 52.7	BOOL	// SLIDE GATE 10-CO2 OPENED
"A_1171_MXZ01_I1"	I 53.0	BOOL	// SLIDE GATE 11-CO2 OPEN
"A_1171_MXZ01_I2"	I 53.1	BOOL	// SLIDE GATE 11-CO2 CLOSE
"A_1171_BZS01_I1"	I 53.2	BOOL	// SLIDE GATE 11-CO2 CLOSED
"A_1171_BZS02_I1"	I 53.3	BOOL	// SLIDE GATE 11-CO2 OPENED
"A_1172_MXZ01_I1"	I 53.4	BOOL	// SLIDE GATE 12-CO2 OPEN
"A_1172_MXZ01_I2"	I 53.5	BOOL	// SLIDE GATE 12-CO2 CLOSE
"A_1172_BZS01_I1"	I 53.6	BOOL	// SLIDE GATE 12-CO2 CLOSED
"A_1172_BZS02_I1"	I 53.7	BOOL	// SLIDE GATE 12-CO2 OPENED
"A_1173_MXZ01_I1"	I 54.0	BOOL	// SLIDE GATE 13-CO2 OPEN
"A_1173_MXZ01_I2"	I 54.1	BOOL	// SLIDE GATE 13-CO2 CLOSE
"A_1173_BZS01_I1"	I 54.2	BOOL	// SLIDE GATE 13-CO2 CLOSED
"A_1173_BZS02_I1"	I 54.3	BOOL	// SLIDE GATE 13-CO2 OPENED
"A_1174_MXZ01_I1"	I 54.4	BOOL	// SLIDE GATE 14-CO2 OPEN
"A_1174_MXZ01_I2"	I 54.5	BOOL	// SLIDE GATE 14-CO2 CLOSE
"A_1174_BZS01_I1"	I 54.6	BOOL	// SLIDE GATE 14-CO2 CLOSED
"A_1174_BZS02_I1"	I 54.7	BOOL	// SLIDE GATE 14-CO2 OPENED
"A_1175_MXZ01_I1"	I 55.0	BOOL	// SLIDE GATE 15-CO2 OPEN
"A_1175_MXZ01_I2"	I 55.1	BOOL	// SLIDE GATE 15-CO2 CLOSE
"A_1175_BZS01_I1"	I 55.2	BOOL	// SLIDE GATE 15-CO2 CLOSED
"A_1175_BZS02_I1"	I 55.3	BOOL	// SLIDE GATE 15-CO2 OPENED
"A_1176_MXZ01_I1"	I 55.4	BOOL	// SLIDE GATE 16-CO2 OPEN
"A_1176_MXZ01_I2"	I 55.5	BOOL	// SLIDE GATE 16-CO2 CLOSE
"A_1176_BZS01_I1"	I 55.6	BOOL	// SLIDE GATE 16-CO2 CLOSED
"A_1176_BZS02_I1"	I 55.7	BOOL	// SLIDE GATE 16-CO2 OPENED
"A_1177_MXZ01_I1"	I 56.0	BOOL	// SLIDE GATE 17-CO2 OPEN
"A_1177_MXZ01_I2"	I 56.1	BOOL	// SLIDE GATE 17-CO2 CLOSE
"A_1177_BZS01_I1"	I 56.2	BOOL	// SLIDE GATE 17-CO2 CLOSED
"A_1177_BZS02_I1"	I 56.3	BOOL	// SLIDE GATE 17-CO2 OPENED
"A_1178_MXZ01_I1"	I 56.4	BOOL	// SLIDE GATE 18-CO2 OPEN
"A_1178_MXZ01_I2"	I 56.5	BOOL	// SLIDE GATE 18-CO2 CLOSE
"A_1178_BZS01_I1"	I 56.6	BOOL	// SLIDE GATE 18-CO2 CLOSED
"A_1178_BZS02_I1"	I 56.7	BOOL	// SLIDE GATE 18-CO2 OPENED
"A_1179_MXZ01_I1"	I 57.0	BOOL	// SLIDE GATE 19-CO2 OPEN
"A_1179_MXZ01_I2"	I 57.1	BOOL	// SLIDE GATE 19-CO2 CLOSE
"A_1179_BZS01_I1"	I 57.2	BOOL	// SLIDE GATE 19-CO2 CLOSED
"A_1179_BZS02_I1"	I 57.3	BOOL	// SLIDE GATE 19-CO2 OPENED
"A_1180_MXZ01_I1"	I 57.4	BOOL	// SLIDE GATE 20-CO2 OPEN
"A_1180_MXZ01_I2"	I 57.5	BOOL	// SLIDE GATE 20-CO2 CLOSE
"A_1180_BZS01_I1"	I 57.6	BOOL	// SLIDE GATE 20-CO2 CLOSED
"A_1180_BZS02_I1"	I 57.7	BOOL	// SLIDE GATE 20-CO2 OPENED
"A_1181_MXZ01_I1"	I 58.0	BOOL	// SLIDE GATE 21-CO2 OPEN
"A_1181_MXZ01_I2"	I 58.1	BOOL	// SLIDE GATE 21-CO2 CLOSE
"A_1181_BZS01_I1"	I 58.2	BOOL	// SLIDE GATE 21-CO2 CLOSED
"A_1181_BZS02_I1"	I 58.3	BOOL	// SLIDE GATE 21-CO2 OPENED
"A_1182_MXZ01_I1"	I 58.4	BOOL	// SLIDE GATE 22-CO2 OPEN
"A_1182_MXZ01_I2"	I 58.5	BOOL	// SLIDE GATE 22-CO2 CLOSE
"A_1182_BZS01_I1"	I 58.6	BOOL	// SLIDE GATE 22-CO2 CLOSED
"A_1182_BZS02_I1"	I 58.7	BOOL	// SLIDE GATE 22-CO2 OPENED
"A_1183_MXZ01_I1"	I 59.0	BOOL	// SLIDE GATE 23-CO2 OPEN
"A_1183_MXZ01_I2"	I 59.1	BOOL	// SLIDE GATE 23-CO2 CLOSE
"A_1183_BZS01_I1"	I 59.2	BOOL	// SLIDE GATE 23-CO2 CLOSED
"A_1183_BZS02_I1"	I 59.3	BOOL	// SLIDE GATE 23-CO2 OPENED
"A_1184_MXZ01_I1"	I 59.4	BOOL	// SLIDE GATE 24-CO2 OPEN
"A_1184_MXZ01_I2"	I 59.5	BOOL	// SLIDE GATE 24-CO2 CLOSE
"A_1184_BZS01_I1"	I 59.6	BOOL	// SLIDE GATE 24-CO2 CLOSED
"A_1184_BZS02_I1"	I 59.7	BOOL	// SLIDE GATE 24-CO2 OPENED
"A_1111_MXZ45_I1"	I 64.0	BOOL	// AERATION-VALVE 1 OPEN
"A_1111_MXZ45_I2"	I 64.1	BOOL	// AERATION-VALVE 1 CLOSE
"A_1111_BZS47_I1"	I 64.2	BOOL	// AERATION-VALVE 1 CLOSED
"A_1111_BZS48_I1"	I 64.3	BOOL	// AERATION-VALVE 1 OPENED
"A_1112_MXZ45_I1"	I 64.4	BOOL	// AERATION-VALVE 2 OPEN
"A_1112_MXZ45_I2"	I 64.5	BOOL	// AERATION-VALVE 2 CLOSE
"A_1112_BZS47_I1"	I 64.6	BOOL	// AERATION-VALVE 2 CLOSED
"A_1112_BZS48_I1"	I 64.7	BOOL	// AERATION-VALVE 2 OPENED
"A_1113_MXZ45_I1"	I 65.0	BOOL	// AERATION-VALVE 3 OPEN
"A_1113_MXZ45_I2"	I 65.1	BOOL	// AERATION-VALVE 3 CLOSE
"A_1113_BZS47_I1"	I 65.2	BOOL	// AERATION-VALVE 3 CLOSED
"A_1113_BZS48_I1"	I 65.3	BOOL	// AERATION-VALVE 3 OPENED
"A_1114_MXZ45_I1"	I 65.4	BOOL	// AERATION-VALVE 4 OPEN
"A_1114_MXZ45_I2"	I 65.5	BOOL	// AERATION-VALVE 4 CLOSE
"A_1114_BZS47_I1"	I 65.6	BOOL	// AERATION-VALVE 4 CLOSED
"A_1114_BZS48_I1"	I 65.7	BOOL	// AERATION-VALVE 4 OPENED
"A_1115_MXZ45_I1"	I 66.0	BOOL	// AERATION-VALVE 5 OPEN
"A_1115_MXZ45_I2"	I 66.1	BOOL	// AERATION-VALVE 5 CLOSE
"A_1115_BZS47_I1"	I 66.2	BOOL	// AERATION-VALVE 5 CLOSED
"A_1115_BZS48_I1"	I 66.3	BOOL	// AERATION-VALVE 5 OPENED
"A_1116_MXZ45_I1"	I 66.4	BOOL	// AERATION-VALVE 6 OPEN
"A_1116_MXZ45_I2"	I 66.5	BOOL	// AERATION-VALVE 6 CLOSE
"A_1116_BZS47_I1"	I 66.6	BOOL	// AERATION-VALVE 6 CLOSED
"A_1116_BZS48_I1"	I 66.7	BOOL	// AERATION-VALVE 6 OPENED
"A_1117_MXZ45_I1"	I 67.0	BOOL	// AERATION-VALVE 7 OPEN
"A_1117_MXZ45_I2"	I 67.1	BOOL	// AERATION-VALVE 7 CLOSE
"A_1117_BZS47_I1"	I 67.2	BOOL	// AERATION-VALVE 7 CLOSED
"A_1117_BZS48_I1"	I 67.3	BOOL	// AERATION-VALVE 7 OPENED
"A_1118_MXZ45_I1"	I 67.4	BOOL	// AERATION-VALVE 8 OPEN
"A_1118_MXZ45_I2"	I 67.5	BOOL	// AERATION-VALVE 8 CLOSE
"A_1118_BZS47_I1"	I 67.6	BOOL	// AERATION-VALVE 8 CLOSED
"A_1118_BZS48_I1"	I 67.7	BOOL	// AERATION-VALVE 8 OPENED
"A_21_A040Z1_I1"	I 100.0	BOOL	// POWER SUPPLY FAILURE +C21
"A_21_S_H097Z1_I1"	I 100.1	BOOL	// OPERATING ON +C21
"A_21_K091Z1_I1"	I 100.2	BOOL	// FUSE SWITCH OFF +C21
"A_21_A097Z1_I1"	I 100.3	BOOL	// EMERGENCY-STOP +C21
"A_21_A098Z1_I1"	I 100.4	BOOL	// EMERGENCY-STOP +M211/M212
"A_21_Q390Z1_I1"	I 100.5	BOOL	// POWER SUPPLY MACHINE BMKE
"A_21_Q445Z1_I1"	I 100.6	BOOL	// POWER SUPPLY MACHINE DBFL
"A_21_D1B065_I1"	I 100.7	BOOL	// CONTROL 24VDC LIMIT SWITCHES WAY
"A_2199_SHE01_I1"	I 101.0	BOOL	// EMERGENCY-OFF CUSTOMER
"A_2199_SHE02_I1"	I 101.1	BOOL	// EMERGENCY-OFF CUSTOMER
"A_21_A700Z1_I1"	I 101.4	BOOL	// POWER CIRCUIT CABLE CHAIN
"A_21_A800Z1_I1"	I 101.6	BOOL	// POWER CIRCUIT CABLE CHAIN
"A_2101_MXZ01_I1"	I 102.0	BOOL	// BELT CONVEYOR
"A_2102_YMXZ01_I1"	I 102.1	BOOL	// CHUTE DRIVE LEFT SIDE
"A_2102_YMXZ01_I2"	I 102.2	BOOL	// CHUTE DRIVE RIGHT SIDE
"A_2111_MXZ41_I1"	I 103.0	BOOL	// TRAVELING DRIVE
"A_2111_MXZ61_I1"	I 103.2	BOOL	// TURNING SCREW DRIVE 1
"A_2111_MXZ62_I1"	I 103.3	BOOL	// TURNING SCREW DRIVE 2
"A_2111_MXZ63_I1"	I 103.4	BOOL	// TURNING SCREW DRIVE 3
"A_2111_MXZ64_I1"	I 103.5	BOOL	// TURNING SCREW DRIVE 4
"A_2111_MXZ65_I1"	I 103.6	BOOL	// TURNING SCREW DRIVE 5
"A_2111_MXZ66_I1"	I 103.7	BOOL	// TURNING SCREW DRIVE 6
"A_2111_MXZ67_I1"	I 104.0	BOOL	// TURNING SCREW DRIVE 7
"A_2111_MXZ68_I1"	I 104.1	BOOL	// TURNING SCREW DRIVE 8
"A_2111_MXZ69_I1"	I 104.2	BOOL	// TURNING SCREW DRIVE 9
"A_2111_MXZ70_I1"	I 104.3	BOOL	// TURNING SCREW DRIVE 10
"A_2111_MXZ71_I1"	I 104.4	BOOL	// TURNING SCREW DRIVE 11
"A_2111_MXZ72_I1"	I 104.5	BOOL	// TURNING SCREW DRIVE 12
"A_2111_MXZ73_I1"	I 104.6	BOOL	// TURNING SCREW DRIVE 13
"A_2101_SHE20_I1"	I 105.0	BOOL	// CABLE PULL SWITCH RIGHT 1
"A_2101_SHE21_I1"	I 105.1	BOOL	// CABLE PULL SWITCH RIGHT 2
"A_2101_SHE22_I1"	I 105.2	BOOL	// CABLE PULL SWITCH LEFT 1
"A_2101_SHE23_I1"	I 105.3	BOOL	// CABLE PULL SWITCH LEFT 2
"A_2102_QYS21_I1"	I 105.5	BOOL	// DISCHARGE CHUTE LEFT SIDE
"A_2102_QYS22_I1"	I 105.6	BOOL	// DISCHARGE CHUTE RIGHT SIDE
"A_2115_MXZ11_I1"	I 108.0	BOOL	// HORIZONTAL SCREW
"A_2115_MXZ15_I1"	I 108.2	BOOL	// LIFTING SCREW
"A_2115_MXZ21_I1"	I 108.3	BOOL	// LIFTING DEVICE DOWN
"A_2115_MXZ21_I2"	I 108.4	BOOL	// LIFTING DEVICE UP
"A_21_A458Z1_I1"	I 110.0	BOOL	// CLEANING FLAP 1/2
"A_2115_BZS22_I1"	I 110.6	BOOL	// LIFTING DEVICE DOWN
"A_2115_BZS23_I1"	I 110.7	BOOL	// LIFTING DEVICE END POSITION TOP
"A_2145_QXV21_I1"	I 116.0	BOOL	// RUNNING COOLING UNIT GERMINATING
"A_2145_QXV31_I1"	I 116.1	BOOL	// RUNNING COOLING UNIT GERMINATING
"A_2116_BZS12_I1"	I 116.4	BOOL	// SPRINKING WATER LINE OPENED
"A_2116_BZS11_I1"	I 116.5	BOOL	// SPRINKING WATER LINE CLOSED
"A_2131_BZS12_I1"	I 117.2	BOOL	// VALVE HUMIDIFICATION OPENED
"A_2131_BZS11_I1"	I 117.3	BOOL	// VALVE HUMIDIFICATION CLOSED
"A_2101_BSA13_I1"	I 117.4	BOOL	// SPEED CONTROL
"A_2101_BZS14_15_I1"	I 117.6	BOOL	// BELT MONITOR RIGHT
"A_2101_BZS16_17_I1"	I 117.7	BOOL	// BELT MONITOR LEFT
"A_2102_BZS13_I1"	I 118.2	BOOL	// DISCHARGE CHUTE PARKING POSITION
"A_2102_BZS14_I1"	I 118.3	BOOL	// DISCHARGE CHUTE LEFT SIDE
"A_2102_BZS15_I1"	I 118.4	BOOL	// DISCHARGE CHUTE RIGHT SIDE
"A_2112_BZS12_I1"	I 140.0	BOOL	// SPRINKING WATER LINE 1 OPENED
"A_2112_BZS11_I1"	I 140.1	BOOL	// SPRINKING WATER LINE 1 CLOSED
"A_2112_BZS22_I1"	I 140.2	BOOL	// SPRINKING WATER LINE 2 OPENED
"A_2112_BZS21_I1"	I 140.3	BOOL	// SPRINKING WATER LINE 2 CLOSED
"A_2111_KCL01_I1"	I 140.4	BOOL	// SCREW ON
"A_2111_KCL01_I2"	I 140.5	BOOL	// SCREW OFF
"A_2111_KCL01_I3"	I 140.6	BOOL	// DRIVE FORWARD SLOWLY
"A_2111_KCL01_I4"	I 140.7	BOOL	// DRIVE BACKWARD SLOWLY
"A_2111_KCL01_I5"	I 141.0	BOOL	// DRIVE FORWARD FASTER
"A_2111_KCL01_I6"	I 141.1	BOOL	// DRIVE BACKWARD FASTER
"A_2111_BZS44_I1"	I 141.2	BOOL	// TRAVELING DRIVE STOP LEFT SIDE
"A_2111_BZS46_I1"	I 141.3	BOOL	// TRAVELING DRIVE STOP RIGHT SIDE
"A_21_K738R1_I1"	I 142.0	BOOL	// FUSE SWITCH OFF +M211
"A_21_A408Z1_I1"	I 142.1	BOOL	// BUMPER SWITCHED-OFF
"A_2199_SHE03_I1"	I 142.2	BOOL	// EMERGENCY-STOP 1 MACHINE BMKE
"A_2199_SHE06_I1"	I 142.3	BOOL	// EMERGENCY-STOP 2 MACHINE BMKE
"A_2111_QYS43_I1"	I 142.4	BOOL	// TRAVELING DRIVE SAFETY STLEFT SIDE
"A_2111_QYS45_I1"	I 142.5	BOOL	// TRAVELING DRIVE SAFETY STRIGHT SIDE
"A_2199_SHE20_I1"	I 142.6	BOOL	// CABLE PULL SWITCH RIGHT
"A_2199_SHE21_I1"	I 142.7	BOOL	// CABLE PULL SWITCH LEFT
"A_2111_BZS22_I1"	I 143.0	BOOL	// COUPLING DRIVE UNLOCKED
"A_2111_BZS23_I1"	I 143.1	BOOL	// COUPLING DRIVE LOCKED
"A_2111_BZS26_I1"	I 143.2	BOOL	// COUPLING DRIVE UNLOCKED
"A_2111_BZS27_I1"	I 143.3	BOOL	// COUPLING DRIVE LOCKED
"A_2111_BZS32_I1"	I 143.4	BOOL	// COUPLING DRIVE UNLOCKED
"A_2111_BZS33_I1"	I 143.5	BOOL	// COUPLING DRIVE LOCKED
"A_2111_BZS36_I1"	I 143.6	BOOL	// COUPLING DRIVE UNLOCKED
"A_2111_BZS37_I1"	I 143.7	BOOL	// COUPLING DRIVE LOCKED
"A_2115_KCL01_I1"	I 160.0	BOOL	// BACKWALL LIFTING
"A_2115_KCL01_I2"	I 160.1	BOOL	// BACKWALL LOWERING
"A_2115_KCL01_I3"	I 160.2	BOOL	// UNCOUPLE
"A_2115_KCL01_I4"	I 160.3	BOOL	// COUPLE
"A_2115_KCL01_I5"	I 160.4	BOOL	// WALL LOCKING
"A_2115_KCL01_I6"	I 160.5	BOOL	// WALL UNLOCKING
"A_2115_KCL01_I7"	I 160.6	BOOL	// HORIZONTAL SCREW ON
"A_2115_KCL01_I8"	I 160.7	BOOL	// DIAGONAL SCREW ON
"A_2115_KCL01_I9"	I 161.0	BOOL	// SCREW STOP
"A_2115_BSA12_I1"	I 161.2	BOOL	// ZERO SPEED MONITOR HORIZONTAL SCREW
"A_2115_BSA17_I1"	I 161.3	BOOL	// ZERO SPEED MONITOR LIFTING SCREW
"A_21_K838R1_I1"	I 162.0	BOOL	// FUSE SWITCH OFF +M212
"A_2199_SHE04_I1"	I 162.1	BOOL	// EMERGENCY-STOP 1 MACHINE DBFL
"A_2199_SHE05_I1"	I 162.2	BOOL	// EMERGENCY-STOP 2 MACHINE DBFL
"A_2199_SHE08_I1"	I 162.3	BOOL	// EMERGENCY-STOP 3 MACHINE DBFL
"A_2115_QYS18_I1"	I 162.4	BOOL	// CLEANING FLAP 1
"A_2115_QYS19_I1"	I 162.5	BOOL	// CLEANING FLAP 2
"A_2115_BTT11_I1"	I 162.6	BOOL	// THERMISTOR HORIZONTAL SCREW
"A_2115_BTT15_I1"	I 162.7	BOOL	// THERMISTOR LIFTING SCREW
"A_2115_BZS42_I1"	I 163.0	BOOL	// COUPLING DRIVE UNLOCKED
"A_2115_BZS43_I1"	I 163.1	BOOL	// COUPLING DRIVE LOCKED
"A_2115_BZS46_I1"	I 163.2	BOOL	// COUPLING DRIVE UNLOCKED
"A_2115_BZS47_I1"	I 163.3	BOOL	// COUPLING DRIVE LOCKED
"A_2150_MXZ01_I1"	I 164.0	BOOL	// AIR-FLAP 1 OPEN
"A_2150_MXZ01_I2"	I 164.1	BOOL	// AIR-FLAP 1 CLOSE
"A_2150_BZS01_I1"	I 164.2	BOOL	// AIR-FLAP 1 CLOSED
"A_2150_BZS02_I1"	I 164.3	BOOL	// AIR-FLAP 1 OPENED
"A_2151_MXZ01_I1"	I 164.4	BOOL	// AIR-FLAP 2 OPEN
"A_2151_MXZ01_I2"	I 164.5	BOOL	// AIR-FLAP 2 CLOSE
"A_2151_BZS01_I1"	I 164.6	BOOL	// AIR-FLAP 2 CLOSED
"A_2151_BZS02_I1"	I 164.7	BOOL	// AIR-FLAP 2 OPENED
"A_2152_MXZ01_I1"	I 165.0	BOOL	// AIR-FLAP 3 OPEN
"A_2152_MXZ01_I2"	I 165.1	BOOL	// AIR-FLAP 3 CLOSE
"A_2152_BZS01_I1"	I 165.2	BOOL	// AIR-FLAP 3 CLOSED
"A_2152_BZS02_I1"	I 165.3	BOOL	// AIR-FLAP 3 OPENED
"A_2154_MXZ01_I1"	I 165.4	BOOL	// WATER PUMP 1
"A_2155_MXZ01_I1"	I 165.5	BOOL	// WATER PUMP 2
"A_2160_MXZ01_I1"	I 165.6	BOOL	// GERM FAN 1
"A_2160_MXZ02_I1"	I 165.7	BOOL	// GERM FAN 2
"A_22_A040Z1_I1"	I 200.0	BOOL	// POWER SUPPLY FAILURE +C22
"A_22_S_H097Z1_I1"	I 200.1	BOOL	// OPERATING ON +C22
"A_22_K091Z1_I1"	I 200.2	BOOL	// FUSE SWITCH OFF +C22
"A_22_A097Z1_I1"	I 200.3	BOOL	// EMERGENCY-STOP +C22
"A_22_A098Z1_I1"	I 200.4	BOOL	// EMERGENCY-STOP +M221/M222
"A_22_Q390Z1_I1"	I 200.5	BOOL	// POWER SUPPLY MACHINE BMKE
"A_22_Q445Z1_I1"	I 200.6	BOOL	// POWER SUPPLY MACHINE DBFL
"A_22_D1B065_I1"	I 200.7	BOOL	// CONTROL 24VDC LIMIT SWITCHES WAY
"A_2299_SHE01_I1"	I 201.0	BOOL	// EMERGENCY-OFF CUSTOMER
"A_2299_SHE02_I1"	I 201.1	BOOL	// EMERGENCY-OFF CUSTOMER
"A_22_A700Z1_I1"	I 201.4	BOOL	// POWER CIRCUIT CABLE CHAIN
"A_22_A800Z1_I1"	I 201.6	BOOL	// POWER CIRCUIT CABLE CHAIN
"A_2201_MXZ01_I1"	I 202.0	BOOL	// BELT CONVEYOR
"A_2202_YMXZ01_I1"	I 202.1	BOOL	// CHUTE DRIVE LEFT SIDE
"A_2202_YMXZ01_I2"	I 202.2	BOOL	// CHUTE DRIVE RIGHT SIDE
"A_2211_MXZ41_I1"	I 203.0	BOOL	// TRAVELING DRIVE
"A_2211_MXZ61_I1"	I 203.2	BOOL	// TURNING SCREW DRIVE 1
"A_2211_MXZ62_I1"	I 203.3	BOOL	// TURNING SCREW DRIVE 2
"A_2211_MXZ64_I1"	I 203.5	BOOL	// TURNING SCREW DRIVE 4
"A_2211_MXZ65_I1"	I 203.6	BOOL	// TURNING SCREW DRIVE 5
"A_2211_MXZ66_I1"	I 203.7	BOOL	// TURNING SCREW DRIVE 6
"A_2211_MXZ67_I1"	I 204.0	BOOL	// TURNING SCREW DRIVE 7
"A_2211_MXZ68_I1"	I 204.1	BOOL	// TURNING SCREW DRIVE 8
"A_2211_MXZ69_I1"	I 204.2	BOOL	// TURNING SCREW DRIVE 9
"A_2211_MXZ70_I1"	I 204.3	BOOL	// TURNING SCREW DRIVE 10
"A_2211_MXZ71_I1"	I 204.4	BOOL	// TURNING SCREW DRIVE 11
"A_2211_MXZ72_I1"	I 204.5	BOOL	// TURNING SCREW DRIVE 12
"A_2211_MXZ73_I1"	I 204.6	BOOL	// TURNING SCREW DRIVE 13
"A_2201_SHE20_I1"	I 205.0	BOOL	// CABLE PULL SWITCH RIGHT 1
"A_2201_SHE21_I1"	I 205.1	BOOL	// CABLE PULL SWITCH RIGHT 2
"A_2201_SHE22_I1"	I 205.2	BOOL	// CABLE PULL SWITCH LEFT 1
"A_2201_SHE23_I1"	I 205.3	BOOL	// CABLE PULL SWITCH LEFT 2
"A_2202_QYS21_I1"	I 205.5	BOOL	// DISCHARGE CHUTE LEFT SIDE
"A_2202_QYS22_I1"	I 205.6	BOOL	// DISCHARGE CHUTE RIGHT SIDE
"A_2215_MXZ11_I1"	I 208.0	BOOL	// HORIZONTAL SCREW
"A_2215_MXZ15_I1"	I 208.2	BOOL	// LIFTING SCREW
"A_2215_MXZ21_I1"	I 208.3	BOOL	// LIFTING DEVICE DOWN
"A_2215_MXZ21_I2"	I 208.4	BOOL	// LIFTING DEVICE UP
"A_22_A458Z1_I1"	I 210.0	BOOL	// CLEANING FLAP 1/2
"A_2215_BZS22_I1"	I 210.6	BOOL	// LIFTING DEVICE DOWN
"A_2215_BZS23_I1"	I 210.7	BOOL	// LIFTING DEVICE END POSITION TOP
"A_2245_QXV21_I1"	I 216.0	BOOL	// RUNNING COOLING UNIT GERMINATING
"A_2245_QXV31_I1"	I 216.1	BOOL	// RUNNING COOLING UNIT GERMINATING
"A_2216_BZS12_I1"	I 216.4	BOOL	// SPRINKING WATER LINE OPENED
"A_2216_BZS11_I1"	I 216.5	BOOL	// SPRINKING WATER LINE CLOSED
"A_2231_BZS12_I1"	I 217.2	BOOL	// VALVE HUMIDIFICATION OPENED
"A_2231_BZS11_I1"	I 217.3	BOOL	// VALVE HUMIDIFICATION CLOSED
"A_2201_BSA13_I1"	I 217.4	BOOL	// SPEED CONTROL
"A_2201_BZS14_15_I1"	I 217.6	BOOL	// BELT MONITOR RIGHT
"A_2201_BZS16_17_I1"	I 217.7	BOOL	// BELT MONITOR LEFT
"A_2202_BZS13_I1"	I 218.2	BOOL	// DISCHARGE CHUTE PARKING POSITION
"A_2202_BZS14_I1"	I 218.3	BOOL	// DISCHARGE CHUTE LEFT SIDE
"A_2202_BZS15_I1"	I 218.4	BOOL	// DISCHARGE CHUTE RIGHT SIDE
"A_2212_BZS12_I1"	I 240.0	BOOL	// SPRINKING WATER LINE 1 OPENED
"A_2212_BZS11_I1"	I 240.1	BOOL	// SPRINKING WATER LINE 1 CLOSED
"A_2212_BZS22_I1"	I 240.2	BOOL	// SPRINKING WATER LINE 2 OPENED
"A_2212_BZS21_I1"	I 240.3	BOOL	// SPRINKING WATER LINE 2 CLOSED
"A_2211_KCL01_I1"	I 240.4	BOOL	// SCREW ON
"A_2211_KCL01_I2"	I 240.5	BOOL	// SCREW OFF
"A_2211_KCL01_I3"	I 240.6	BOOL	// DRIVE FORWARD SLOWLY
"A_2211_KCL01_I4"	I 240.7	BOOL	// DRIVE BACKWARD SLOWLY
"A_2211_KCL01_I5"	I 241.0	BOOL	// DRIVE FORWARD FASTER
"A_2211_KCL01_I6"	I 241.1	BOOL	// DRIVE BACKWARD FASTER
"A_2211_BZS44_I1"	I 241.2	BOOL	// TRAVELING DRIVE STOP LEFT SIDE
"A_2211_BZS46_I1"	I 241.3	BOOL	// TRAVELING DRIVE STOP RIGHT SIDE
"A_22_K738R1_I1"	I 242.0	BOOL	// FUSE SWITCH OFF +M221
"A_22_A408Z1_I1"	I 242.1	BOOL	// BUMPER SWITCHED-OFF
"A_2299_SHE03_I1"	I 242.2	BOOL	// EMERGENCY-STOP 1 MACHINE BMKE
"A_2299_SHE06_I1"	I 242.3	BOOL	// EMERGENCY-STOP 2 MACHINE BMKE
"A_2211_QYS43_I1"	I 242.4	BOOL	// TRAVELING DRIVE SAFETY STLEFT SIDE
"A_2211_QYS45_I1"	I 242.5	BOOL	// TRAVELING DRIVE SAFETY STRIGHT SIDE
"A_2299_SHE20_I1"	I 242.6	BOOL	// CABLE PULL SWITCH RIGHT
"A_2299_SHE21_I1"	I 242.7	BOOL	// CABLE PULL SWITCH LEFT
"A_2211_BZS22_I1"	I 243.0	BOOL	// COUPLING DRIVE UNLOCKED
"A_2211_BZS23_I1"	I 243.1	BOOL	// COUPLING DRIVE LOCKED
"A_2211_BZS26_I1"	I 243.2	BOOL	// COUPLING DRIVE UNLOCKED
"A_2211_BZS27_I1"	I 243.3	BOOL	// COUPLING DRIVE LOCKED
"A_2211_BZS32_I1"	I 243.4	BOOL	// COUPLING DRIVE UNLOCKED
"A_2211_BZS33_I1"	I 243.5	BOOL	// COUPLING DRIVE LOCKED
"A_2211_BZS36_I1"	I 243.6	BOOL	// COUPLING DRIVE UNLOCKED
"A_2211_BZS37_I1"	I 243.7	BOOL	// COUPLING DRIVE LOCKED
"A_2215_KCL01_I1"	I 260.0	BOOL	// BACKWALL LIFTING
"A_2215_KCL01_I2"	I 260.1	BOOL	// BACKWALL LOWERING
"A_2215_KCL01_I3"	I 260.2	BOOL	// UNCOUPLE
"A_2215_KCL01_I4"	I 260.3	BOOL	// COUPLE
"A_2215_KCL01_I5"	I 260.4	BOOL	// WALL LOCKING
"A_2215_KCL01_I6"	I 260.5	BOOL	// WALL UNLOCKING
"A_2215_KCL01_I7"	I 260.6	BOOL	// HORIZONTAL SCREW ON
"A_2215_KCL01_I8"	I 260.7	BOOL	// DIAGONAL SCREW ON
"A_2215_KCL01_I9"	I 261.0	BOOL	// SCREW STOP
"A_2215_BSA12_I1"	I 261.2	BOOL	// ZERO SPEED MONITOR HORIZONTAL SCREW
"A_2215_BSA17_I1"	I 261.3	BOOL	// ZERO SPEED MONITOR LIFTING SCREW
"A_22_K838R1_I1"	I 262.0	BOOL	// FUSE SWITCH OFF +M222
"A_2299_SHE04_I1"	I 262.1	BOOL	// EMERGENCY-STOP 1 MACHINE DBFL
"A_2299_SHE05_I1"	I 262.2	BOOL	// EMERGENCY-STOP 2 MACHINE DBFL
"A_2299_SHE08_I1"	I 262.3	BOOL	// EMERGENCY-STOP 3 MACHINE DBFL
"A_2215_QYS18_I1"	I 262.4	BOOL	// CLEANING FLAP 1
"A_2215_QYS19_I1"	I 262.5	BOOL	// CLEANING FLAP 2
"A_2215_BTT11_I1"	I 262.6	BOOL	// THERMISTOR HORIZONTAL SCREW
"A_2215_BTT15_I1"	I 262.7	BOOL	// THERMISTOR LIFTING SCREW
"A_2215_BZS42_I1"	I 263.0	BOOL	// COUPLING DRIVE UNLOCKED
"A_2215_BZS43_I1"	I 263.1	BOOL	// COUPLING DRIVE LOCKED
"A_2215_BZS46_I1"	I 263.2	BOOL	// COUPLING DRIVE UNLOCKED
"A_2215_BZS47_I1"	I 263.3	BOOL	// COUPLING DRIVE LOCKED
"A_2250_MXZ01_I1"	I 264.0	BOOL	// AIR-FLAP 1 OPEN
"A_2250_MXZ01_I2"	I 264.1	BOOL	// AIR-FLAP 1 CLOSE
"A_2250_BZS01_I1"	I 264.2	BOOL	// AIR-FLAP 1 CLOSED
"A_2250_BZS02_I1"	I 264.3	BOOL	// AIR-FLAP 1 OPENED
"A_2251_MXZ01_I1"	I 264.4	BOOL	// AIR-FLAP 2 OPEN
"A_2251_MXZ01_I2"	I 264.5	BOOL	// AIR-FLAP 2 CLOSE
"A_2251_BZS01_I1"	I 264.6	BOOL	// AIR-FLAP 2 CLOSED
"A_2251_BZS02_I1"	I 264.7	BOOL	// AIR-FLAP 2 OPENED
"A_2252_MXZ01_I1"	I 265.0	BOOL	// AIR-FLAP 3 OPEN
"A_2252_MXZ01_I2"	I 265.1	BOOL	// AIR-FLAP 3 CLOSE
"A_2252_BZS01_I1"	I 265.2	BOOL	// AIR-FLAP 3 CLOSED
"A_2252_BZS02_I1"	I 265.3	BOOL	// AIR-FLAP 3 OPENED
"A_2254_MXZ01_I1"	I 265.4	BOOL	// WATER PUMP 1
"A_2255_MXZ01_I1"	I 265.5	BOOL	// WATER PUMP 2
"A_2260_MXZ01_I1"	I 265.6	BOOL	// GERM FAN 1
"A_2260_MXZ02_I1"	I 265.7	BOOL	// GERM FAN 2
"A_23_A040Z1_I1"	I 300.0	BOOL	// POWER SUPPLY FAILURE +C23
"A_23_S_H097Z1_I1"	I 300.1	BOOL	// OPERATING ON +C23
"A_23_K091Z1_I1"	I 300.2	BOOL	// FUSE SWITCH OFF +C23
"A_23_A097Z1_I1"	I 300.3	BOOL	// EMERGENCY-STOP +C23
"A_23_A098Z1_I1"	I 300.4	BOOL	// EMERGENCY-STOP +M231/M232
"A_23_Q390Z1_I1"	I 300.5	BOOL	// POWER SUPPLY MACHINE BMKE
"A_23_Q445Z1_I1"	I 300.6	BOOL	// POWER SUPPLY MACHINE DBFL
"A_23_D1B065_I1"	I 300.7	BOOL	// CONTROL 24VDC LIMIT SWITCHES WAY
"A_2399_SHE01_I1"	I 301.0	BOOL	// EMERGENCY-OFF CUSTOMER
"A_2399_SHE02_I1"	I 301.1	BOOL	// EMERGENCY-OFF CUSTOMER
"A_23_A700Z1_I1"	I 301.4	BOOL	// POWER CIRCUIT CABLE CHAIN
"A_23_A800Z1_I1"	I 301.6	BOOL	// POWER CIRCUIT CABLE CHAIN
"A_2301_MXZ01_I1"	I 302.0	BOOL	// BELT CONVEYOR
"A_2302_YMXZ01_I1"	I 302.1	BOOL	// CHUTE DRIVE LEFT SIDE
"A_2302_YMXZ01_I2"	I 302.2	BOOL	// CHUTE DRIVE RIGHT SIDE
"A_2311_MXZ41_I1"	I 303.0	BOOL	// TRAVELING DRIVE
"A_2311_MXZ61_I1"	I 303.2	BOOL	// TURNING SCREW DRIVE 1
"A_2311_MXZ62_I1"	I 303.3	BOOL	// TURNING SCREW DRIVE 2
"A_2311_MXZ63_I1"	I 303.4	BOOL	// TURNING SCREW DRIVE 3
"A_2311_MXZ64_I1"	I 303.5	BOOL	// TURNING SCREW DRIVE 4
"A_2311_MXZ65_I1"	I 303.6	BOOL	// TURNING SCREW DRIVE 5
"A_2311_MXZ66_I1"	I 303.7	BOOL	// TURNING SCREW DRIVE 6
"A_2311_MXZ67_I1"	I 304.0	BOOL	// TURNING SCREW DRIVE 7
"A_2311_MXZ68_I1"	I 304.1	BOOL	// TURNING SCREW DRIVE 8
"A_2311_MXZ69_I1"	I 304.2	BOOL	// TURNING SCREW DRIVE 9
"A_2311_MXZ70_I1"	I 304.3	BOOL	// TURNING SCREW DRIVE 10
"A_2311_MXZ72_I1"	I 304.5	BOOL	// TURNING SCREW DRIVE 12
"A_2311_MXZ73_I1"	I 304.6	BOOL	// TURNING SCREW DRIVE 13
"A_2301_SHE20_I1"	I 305.0	BOOL	// CABLE PULL SWITCH RIGHT 1
"A_2301_SHE21_I1"	I 305.1	BOOL	// CABLE PULL SWITCH RIGHT 2
"A_2301_SHE22_I1"	I 305.2	BOOL	// CABLE PULL SWITCH LEFT 1
"A_2302_QYS21_I1"	I 305.5	BOOL	// DISCHARGE CHUTE LEFT SIDE
"A_2302_QYS22_I1"	I 305.6	BOOL	// DISCHARGE CHUTE RIGHT SIDE
"A_2315_MXZ11_I1"	I 308.0	BOOL	// HORIZONTAL SCREW
"A_2315_MXZ15_I1"	I 308.2	BOOL	// LIFTING SCREW
"A_2315_MXZ21_I1"	I 308.3	BOOL	// LIFTING DEVICE DOWN
"A_2315_MXZ21_I2"	I 308.4	BOOL	// LIFTING DEVICE UP
"A_23_A458Z1_I1"	I 310.0	BOOL	// CLEANING FLAP 1/2
"A_2315_BZS22_I1"	I 310.6	BOOL	// LIFTING DEVICE DOWN
"A_2315_BZS23_I1"	I 310.7	BOOL	// LIFTING DEVICE END POSITION TOP
"A_2345_QXV21_I1"	I 316.0	BOOL	// RUNNING COOLING UNIT GERMINATING
"A_2345_QXV31_I1"	I 316.1	BOOL	// RUNNING COOLING UNIT GERMINATING
"A_2316_BZS12_I1"	I 316.4	BOOL	// SPRINKING WATER LINE OPENED
"A_2316_BZS11_I1"	I 316.5	BOOL	// SPRINKING WATER LINE CLOSED
"A_2331_BZS12_I1"	I 317.2	BOOL	// VALVE HUMIDIFICATION OPENED
"A_2331_BZS11_I1"	I 317.3	BOOL	// VALVE HUMIDIFICATION CLOSED
"A_2301_BSA13_I1"	I 317.4	BOOL	// SPEED CONTROL
"A_2301_BZS14_15_I1"	I 317.6	BOOL	// BELT MONITOR RIGHT
"A_2301_BZS16_17_I1"	I 317.7	BOOL	// BELT MONITOR LEFT
"A_2302_BZS13_I1"	I 318.2	BOOL	// DISCHARGE CHUTE PARKING POSITION
"A_2302_BZS14_I1"	I 318.3	BOOL	// DISCHARGE CHUTE LEFT SIDE
"A_2302_BZS15_I1"	I 318.4	BOOL	// DISCHARGE CHUTE RIGHT SIDE
"A_2312_BZS12_I1"	I 340.0	BOOL	// SPRINKING WATER LINE 1 OPENED
"A_2312_BZS11_I1"	I 340.1	BOOL	// SPRINKING WATER LINE 1 CLOSED
"A_2312_BZS22_I1"	I 340.2	BOOL	// SPRINKING WATER LINE 2 OPENED
"A_2312_BZS21_I1"	I 340.3	BOOL	// SPRINKING WATER LINE 2 CLOSED
"A_2311_KCL01_I1"	I 340.4	BOOL	// SCREW ON
"A_2311_KCL01_I2"	I 340.5	BOOL	// SCREW OFF
"A_2311_KCL01_I3"	I 340.6	BOOL	// DRIVE FORWARD SLOWLY
"A_2311_KCL01_I4"	I 340.7	BOOL	// DRIVE BACKWARD SLOWLY
"A_2311_KCL01_I5"	I 341.0	BOOL	// DRIVE FORWARD FASTER
"A_2311_KCL01_I6"	I 341.1	BOOL	// DRIVE BACKWARD FASTER
"A_2311_BZS44_I1"	I 341.2	BOOL	// TRAVELING DRIVE STOP LEFT SIDE
"A_2311_BZS46_I1"	I 341.3	BOOL	// TRAVELING DRIVE STOP RIGHT SIDE
"A_23_K738R1_I1"	I 342.0	BOOL	// FUSE SWITCH OFF +M231
"A_23_A408Z1_I1"	I 342.1	BOOL	// BUMPER SWITCHED-OFF
"A_2399_SHE03_I1"	I 342.2	BOOL	// EMERGENCY-STOP 1 MACHINE BMKE
"A_2399_SHE06_I1"	I 342.3	BOOL	// EMERGENCY-STOP 2 MACHINE BMKE
"A_2311_QYS43_I1"	I 342.4	BOOL	// TRAVELING DRIVE SAFETY STLEFT SIDE
"A_2311_QYS45_I1"	I 342.5	BOOL	// TRAVELING DRIVE SAFETY STRIGHT SIDE
"A_2399_SHE20_I1"	I 342.6	BOOL	// CABLE PULL SWITCH RIGHT
"A_2399_SHE21_I1"	I 342.7	BOOL	// CABLE PULL SWITCH LEFT
"A_2311_BZS22_I1"	I 343.0	BOOL	// COUPLING DRIVE UNLOCKED
"A_2311_BZS23_I1"	I 343.1	BOOL	// COUPLING DRIVE LOCKED
"A_2311_BZS26_I1"	I 343.2	BOOL	// COUPLING DRIVE UNLOCKED
"A_2311_BZS27_I1"	I 343.3	BOOL	// COUPLING DRIVE LOCKED
"A_2311_BZS32_I1"	I 343.4	BOOL	// COUPLING DRIVE UNLOCKED
"A_2311_BZS33_I1"	I 343.5	BOOL	// COUPLING DRIVE LOCKED
"A_2311_BZS36_I1"	I 343.6	BOOL	// COUPLING DRIVE UNLOCKED
"A_2311_BZS37_I1"	I 343.7	BOOL	// COUPLING DRIVE LOCKED
"A_2315_KCL01_I1"	I 360.0	BOOL	// BACKWALL LIFTING
"A_2315_KCL01_I2"	I 360.1	BOOL	// BACKWALL LOWERING
"A_2315_KCL01_I3"	I 360.2	BOOL	// UNCOUPLE
"A_2315_KCL01_I4"	I 360.3	BOOL	// COUPLE
"A_2315_KCL01_I5"	I 360.4	BOOL	// WALL LOCKING
"A_2315_KCL01_I6"	I 360.5	BOOL	// WALL UNLOCKING
"A_2315_KCL01_I7"	I 360.6	BOOL	// HORIZONTAL SCREW ON
"A_2315_KCL01_I8"	I 360.7	BOOL	// DIAGONAL SCREW ON
"A_2315_KCL01_I9"	I 361.0	BOOL	// SCREW STOP
"A_2315_BSA12_I1"	I 361.2	BOOL	// ZERO SPEED MONITOR HORIZONTAL SCREW
"A_2315_BSA17_I1"	I 361.3	BOOL	// ZERO SPEED MONITOR LIFTING SCREW
"A_23_K838R1_I1"	I 362.0	BOOL	// FUSE SWITCH OFF +M232
"A_2399_SHE04_I1"	I 362.1	BOOL	// EMERGENCY-STOP 1 MACHINE DBFL
"A_2399_SHE05_I1"	I 362.2	BOOL	// EMERGENCY-STOP 2 MACHINE DBFL
"A_2399_SHE08_I1"	I 362.3	BOOL	// EMERGENCY-STOP 3 MACHINE DBFL
"A_2315_QYS18_I1"	I 362.4	BOOL	// CLEANING FLAP 1
"A_2315_QYS19_I1"	I 362.5	BOOL	// CLEANING FLAP 2
"A_2315_BTT11_I1"	I 362.6	BOOL	// THERMISTOR HORIZONTAL SCREW
"A_2315_BTT15_I1"	I 362.7	BOOL	// THERMISTOR LIFTING SCREW
"A_2315_BZS42_I1"	I 363.0	BOOL	// COUPLING DRIVE UNLOCKED
"A_2315_BZS43_I1"	I 363.1	BOOL	// COUPLING DRIVE LOCKED
"A_2315_BZS46_I1"	I 363.2	BOOL	// COUPLING DRIVE UNLOCKED
"A_2315_BZS47_I1"	I 363.3	BOOL	// COUPLING DRIVE LOCKED
"A_2350_MXZ01_I1"	I 364.0	BOOL	// AIR-FLAP 1 OPEN
"A_2350_MXZ01_I2"	I 364.1	BOOL	// AIR-FLAP 1 CLOSE
"A_2350_BZS01_I1"	I 364.2	BOOL	// AIR-FLAP 1 CLOSED
"A_2350_BZS02_I1"	I 364.3	BOOL	// AIR-FLAP 1 OPENED
"A_2351_MXZ01_I1"	I 364.4	BOOL	// AIR-FLAP 2 OPEN
"A_2351_MXZ01_I2"	I 364.5	BOOL	// AIR-FLAP 2 CLOSE
"A_2351_BZS01_I1"	I 364.6	BOOL	// AIR-FLAP 2 CLOSED
"A_2351_BZS02_I1"	I 364.7	BOOL	// AIR-FLAP 2 OPENED
"A_2352_MXZ01_I1"	I 365.0	BOOL	// AIR-FLAP 3 OPEN
"A_2352_MXZ01_I2"	I 365.1	BOOL	// AIR-FLAP 3 CLOSE
"A_2352_BZS01_I1"	I 365.2	BOOL	// AIR-FLAP 3 CLOSED
"A_2352_BZS02_I1"	I 365.3	BOOL	// AIR-FLAP 3 OPENED
"A_2354_MXZ01_I1"	I 365.4	BOOL	// WATER PUMP 1
"A_2355_MXZ01_I1"	I 365.5	BOOL	// WATER PUMP 2
"A_2360_MXZ01_I1"	I 365.6	BOOL	// GERM FAN 1
"A_2360_MXZ02_I1"	I 365.7	BOOL	// GERM FAN 2
"A_24_A040Z1_I1"	I 400.0	BOOL	// POWER SUPPLY FAILURE +C24
"A_24_S_H097Z1_I1"	I 400.1	BOOL	// OPERATING ON +C24
"A_24_K091Z1_I1"	I 400.2	BOOL	// FUSE SWITCH OFF +C24
"A_24_A097Z1_I1"	I 400.3	BOOL	// EMERGENCY-STOP +C24
"A_24_A098Z1_I1"	I 400.4	BOOL	// EMERGENCY-STOP +M241/M242
"A_24_Q445Z1_I1"	I 400.6	BOOL	// POWER SUPPLY MACHINE DBFL
"A_24_D1B065_I1"	I 400.7	BOOL	// CONTROL 24VDC LIMIT SWITCHES WAY
"A_2499_SHE01_I1"	I 401.0	BOOL	// EMERGENCY-OFF CUSTOMER
"A_2499_SHE02_I1"	I 401.1	BOOL	// EMERGENCY-OFF CUSTOMER
"A_24_A700Z1_I1"	I 401.4	BOOL	// POWER CIRCUIT CABLE CHAIN
"A_24_A800Z1_I1"	I 401.6	BOOL	// POWER CIRCUIT CABLE CHAIN
"A_2401_MXZ01_I1"	I 402.0	BOOL	// BELT CONVEYOR
"A_2402_YMXZ01_I1"	I 402.1	BOOL	// CHUTE DRIVE LEFT SIDE
"A_2402_YMXZ01_I2"	I 402.2	BOOL	// CHUTE DRIVE RIGHT SIDE
"A_2411_MXZ41_I1"	I 403.0	BOOL	// TRAVELING DRIVE
"A_2411_MXZ61_I1"	I 403.2	BOOL	// TURNING SCREW DRIVE 1
"A_2411_MXZ62_I1"	I 403.3	BOOL	// TURNING SCREW DRIVE 2
"A_2411_MXZ63_I1"	I 403.4	BOOL	// TURNING SCREW DRIVE 3
"A_2411_MXZ64_I1"	I 403.5	BOOL	// TURNING SCREW DRIVE 4
"A_2411_MXZ65_I1"	I 403.6	BOOL	// TURNING SCREW DRIVE 5
"A_2411_MXZ66_I1"	I 403.7	BOOL	// TURNING SCREW DRIVE 6
"A_2411_MXZ67_I1"	I 404.0	BOOL	// TURNING SCREW DRIVE 7
"A_2411_MXZ68_I1"	I 404.1	BOOL	// TURNING SCREW DRIVE 8
"A_2411_MXZ69_I1"	I 404.2	BOOL	// TURNING SCREW DRIVE 9
"A_2411_MXZ70_I1"	I 404.3	BOOL	// TURNING SCREW DRIVE 10
"A_2411_MXZ71_I1"	I 404.4	BOOL	// TURNING SCREW DRIVE 11
"A_2411_MXZ72_I1"	I 404.5	BOOL	// TURNING SCREW DRIVE 12
"A_2411_MXZ73_I1"	I 404.6	BOOL	// TURNING SCREW DRIVE 13
"A_2401_SHE20_I1"	I 405.0	BOOL	// CABLE PULL SWITCH RIGHT 1
"A_2401_SHE21_I1"	I 405.1	BOOL	// CABLE PULL SWITCH RIGHT 2
"A_2401_SHE22_I1"	I 405.2	BOOL	// CABLE PULL SWITCH LEFT 1
"A_2401_SHE23_I1"	I 405.3	BOOL	// CABLE PULL SWITCH LEFT 2
"A_2402_QYS21_I1"	I 405.5	BOOL	// DISCHARGE CHUTE LEFT SIDE
"A_2402_QYS22_I1"	I 405.6	BOOL	// DISCHARGE CHUTE RIGHT SIDE
"A_2415_MXZ11_I1"	I 408.0	BOOL	// HORIZONTAL SCREW
"A_2415_MXZ15_I1"	I 408.2	BOOL	// LIFTING SCREW
"A_2415_MXZ21_I1"	I 408.3	BOOL	// LIFTING DEVICE DOWN
"A_2415_MXZ21_I2"	I 408.4	BOOL	// LIFTING DEVICE UP
"A_24_A458Z1_I1"	I 410.0	BOOL	// CLEANING FLAP 1/2
"A_2415_BZS22_I1"	I 410.6	BOOL	// LIFTING DEVICE DOWN
"A_2415_BZS23_I1"	I 410.7	BOOL	// LIFTING DEVICE END POSITION TOP
